FUNCTION_BLOCK "FB_DigitalOutputs"   // FB212, SCL
{ S7_Optimized_Access := 'TRUE' }
// stored: AutoNumber false, MemoryReserve 100, SetENOAutomatically false
   VAR
      sFreeQ0_0 : "FB_DigitalOutput";
      sOperatingCounter : "FB_DigitalOutput";
      sGeneralAirValve : "FB_DigitalOutput";
      sSmartLineDisable : "FB_DigitalOutput";
      sMachineLight : "FB_DigitalOutput";
      sMachineLightBack : "FB_DigitalOutput";
      sLightTowerOrange : "FB_DigitalOutput";
      sLightTowerRed : "FB_DigitalOutput";
      sLightTowerBlue : "FB_DigitalOutput";
      sLightTowerGreen : "FB_DigitalOutput";
      sLightTowerWhite : "FB_DigitalOutput";
      sBacklight : "FB_DigitalOutput";
      sFreeQ1_4 : "FB_DigitalOutput";
      sInfeedON : "FB_DigitalOutput";
      sAxisActivation : "FB_DigitalOutput";
      sBuzzerActivation : "FB_DigitalOutput";
      sElbaronPowerON : "FB_DigitalOutput";
      sObservationCameraLight : "FB_DigitalOutput";
      sLaserExternalDoorOpening : "FB_DigitalOutput";
      sCoolingStart : "FB_DigitalOutput";
      sX_AxisBrakeActivation : "FB_DigitalOutput";
      sY_AxisBrakeActivation : "FB_DigitalOutput";
      sAxisB_TeachInClampingPart : "FB_DigitalOutput";
      sEPO_UPS : "FB_DigitalOutput";
      sHeadLaserStart : "FB_DigitalOutput";
      sHeadLaserStop : "FB_DigitalOutput";
      sAxis2_PowerContactor : "FB_DigitalOutput";
      sGasAssistOn : "FB_DigitalOutput";
      sSmartLineReset : "FB_DigitalOutput";
      sXY_AxisPowerContactor : "FB_DigitalOutput";
      sLaserAirPressureProcess : "FB_DigitalOutput";
      sBus60V_PowerContactor : "FB_DigitalOutput";
      sFreeQ4_0 : "FB_DigitalOutput";
      sFreeQ4_1 : "FB_DigitalOutput";
      sFreeQ4_2 : "FB_DigitalOutput";
      sFreeQ4_3 : "FB_DigitalOutput";
      sLoadClampClosing : "FB_DigitalOutput";
      sLoadClampOpening : "FB_DigitalOutput";
      sUnloadClampClosing : "FB_DigitalOutput";
      sUnloadClampOpening : "FB_DigitalOutput";
      sClampingOpening : "FB_DigitalOutput";
      sClampingClosing : "FB_DigitalOutput";
      sB_AxisBrakeRelease : "FB_DigitalOutput";
      sSuction : "FB_DigitalOutput";
      sFreeQ5_4 : "FB_DigitalOutput";
      sFreeQ5_5 : "FB_DigitalOutput";
      sFreeQ5_6 : "FB_DigitalOutput";
      sFreeQ5_7 : "FB_DigitalOutput";
      sExternalGateClosing : "FB_DigitalOutput";
      sExternalGateOpening : "FB_DigitalOutput";
      sInternalGateClosing : "FB_DigitalOutput";
      sInternalGateOpening : "FB_DigitalOutput";
      sPowerMeterRetract : "FB_DigitalOutput";
      sPowerMeterAdvance : "FB_DigitalOutput";
      sBlowing : "FB_DigitalOutput";
      sFreeQ8_7 : "FB_DigitalOutput";
      sFreeQ9_0 : "FB_DigitalOutput";
      sFreeQ9_1 : "FB_DigitalOutput";
      sFreeQ9_2 : "FB_DigitalOutput";
      sFreeQ9_3 : "FB_DigitalOutput";
      sFreeQ9_4 : "FB_DigitalOutput";
      sFreeQ9_5 : "FB_DigitalOutput";
      sFreeQ9_6 : "FB_DigitalOutput";
      sFreeQ9_7 : "FB_DigitalOutput";
      sSonplasDiagDPCoupler { S7_SetPoint := 'True'} : "FB_DigitalOutput";
      sSonplasReady { S7_SetPoint := 'True'} : "FB_DigitalOutput";
      sSonplasNoEStop { S7_SetPoint := 'True'} : "FB_DigitalOutput";
      sSonplasDoorsClosed { S7_SetPoint := 'True'} : "FB_DigitalOutput";
      sSonplasRunError { S7_SetPoint := 'True'} : "FB_DigitalOutput";
      sSonplasFreeQ200_5 { S7_SetPoint := 'True'} : "FB_DigitalOutput";
      sSonplasFreeQ200_6 { S7_SetPoint := 'True'} : "FB_DigitalOutput";
      sSonplasFreeQ200_7 { S7_SetPoint := 'True'} : "FB_DigitalOutput";
      sSonplasFreeQ201_0 { S7_SetPoint := 'True'} : "FB_DigitalOutput";
      sSonplasFreeQ201_1 { S7_SetPoint := 'True'} : "FB_DigitalOutput";
      sSonplasFreeQ201_2 { S7_SetPoint := 'True'} : "FB_DigitalOutput";
      sSonplasFreeQ201_3 { S7_SetPoint := 'True'} : "FB_DigitalOutput";
      sSonplasFreeQ201_4 { S7_SetPoint := 'True'} : "FB_DigitalOutput";
      sSonplasFreeQ201_5 { S7_SetPoint := 'True'} : "FB_DigitalOutput";
      sSonplasFreeQ201_6 { S7_SetPoint := 'True'} : "FB_DigitalOutput";
      sSonplasFreeQ201_7 { S7_SetPoint := 'True'} : "FB_DigitalOutput";
      sSonplasShuttle1InPos { S7_SetPoint := 'True'} : "FB_DigitalOutput";
      sSonplasFreeQ202_1 { S7_SetPoint := 'True'} : "FB_DigitalOutput";
      sSonplasFreeQ202_2 { S7_SetPoint := 'True'} : "FB_DigitalOutput";
      sSonplasFreeQ202_3 { S7_SetPoint := 'True'} : "FB_DigitalOutput";
      sSonplasFreeQ202_4 { S7_SetPoint := 'True'} : "FB_DigitalOutput";
      sSonplasFreeQ202_5 { S7_SetPoint := 'True'} : "FB_DigitalOutput";
      sSonplasPart1OK { S7_SetPoint := 'True'} : "FB_DigitalOutput";
      sSonplasPart1NOK { S7_SetPoint := 'True'} : "FB_DigitalOutput";
      sSonplasShuttle2InPos { S7_SetPoint := 'True'} : "FB_DigitalOutput";
      sSonplasFreeQ203_1 { S7_SetPoint := 'True'} : "FB_DigitalOutput";
      sSonplasFreeQ203_2 { S7_SetPoint := 'True'} : "FB_DigitalOutput";
      sSonplasFreeQ203_3 { S7_SetPoint := 'True'} : "FB_DigitalOutput";
      sSonplasFreeQ203_4 { S7_SetPoint := 'True'} : "FB_DigitalOutput";
      sSonplasFreeQ203_5 { S7_SetPoint := 'True'} : "FB_DigitalOutput";
      sSonplasPart2OK { S7_SetPoint := 'True'} : "FB_DigitalOutput";
      sSonplasPart2NOK { S7_SetPoint := 'True'} : "FB_DigitalOutput";
      sSonplasResultAccepted { S7_SetPoint := 'True'} : "FB_DigitalOutput";
      sSonplasFreeQ244_1 { S7_SetPoint := 'True'} : "FB_DigitalOutput";
      sSonplasFreeQ244_2 { S7_SetPoint := 'True'} : "FB_DigitalOutput";
      sSonplasFreeQ244_3 { S7_SetPoint := 'True'} : "FB_DigitalOutput";
      sSonplasFreeQ244_4 { S7_SetPoint := 'True'} : "FB_DigitalOutput";
      sSonplasFreeQ244_5 { S7_SetPoint := 'True'} : "FB_DigitalOutput";
      sSonplasFreeQ244_6 { S7_SetPoint := 'True'} : "FB_DigitalOutput";
      sSonplasFreeQ244_7 { S7_SetPoint := 'True'} : "FB_DigitalOutput";
   END_VAR
BEGIN
   REGION Description head
       //==================================================================================
       // POSALUX Swiss SA / (C) Copyright 2025
       //----------------------------------------------------------------------------------
       // Title: Digital Ouputs mapping
       // Comment/Function: Digital Ouputs mapping
       // Author: Fabien WALDT
       // Engineering: TIA Portal v17
       //----------------------------------------------------------------------------------
       // Change log table:
       // Version  | Date     | Expert in charge | Changes applied
       //----------------------------------------------------------------------------------
       // 00.00.01 | 20250423 | WFA              | First released version
       //==================================================================================
   END_REGION


       // ET200SP Mapping
   REGION Q0.0 - Q1.7 : DQ 16x24VDC/0.5A ST Slot 5
       #sFreeQ0_0(oHWStatus => "DQ_FreeQ0_0");
       #sOperatingCounter(oHWStatus => "DQ_OperatingCounter");
       #sGeneralAirValve(oHWStatus => "DQ_GeneralAirValve");
       #sSmartLineDisable(oHWStatus => "DQ_SmartLineDisable");
       #sMachineLight(oHWStatus => "DQ_MachineLight");
       #sMachineLightBack(oHWStatus => "DQ_MachineLightBack");
       #sLightTowerOrange(oHWStatus => "DQ_LightTowerOrange");
       #sLightTowerRed(oHWStatus => "DQ_LightTowerRed");
       //
       #sLightTowerBlue(oHWStatus => "DQ_LightTowerBlue");
       #sLightTowerGreen(oHWStatus => "DQ_Light_owerGreen");
       #sLightTowerWhite(oHWStatus => "DQ_LightTowerWhite");
       #sBacklight(oHWStatus => "DQ_Backlight");
       #sFreeQ1_4(oHWStatus => "DQ_FreeQ1_4");
       #sInfeedON(oHWStatus => "DQ_InfeedON");
       #sAxisActivation(oHWStatus => "DQ_AxisActivation");
       #sBuzzerActivation(oHWStatus => "DQ_BuzzerActivation");
   END_REGION

   REGION Q2.0 - Q3.7 : DQ 16x24VDC/0.5A ST Slot 6
       #sElbaronPowerON(oHWStatus => "DQ_ElbaronPowerON");
       #sObservationCameraLight(oHWStatus => "DQ_ObservationCameraLight");
       #sLaserExternalDoorOpening(oHWStatus => "DQ_LaserExternalDoorOpening");
       #sCoolingStart(oHWStatus => "DQ_CoolingStart");
       #sX_AxisBrakeActivation(oHWStatus => "DQ_X_AxisBrakeActivation");
       #sY_AxisBrakeActivation(oHWStatus => "DQ_Y_AxisBrakeActivation");
       #sAxisB_TeachInClampingPart(oHWStatus => "DQ_AxisB_TeachInClampingPart");
       #sEPO_UPS(oHWStatus => "DQ_EPO_UPS");
       //
       #sHeadLaserStart(oHWStatus => "DQ_HeadLaserStart");
       #sHeadLaserStop(oHWStatus => "DQ_HeadLaserStop");
       #sAxis2_PowerContactor(oHWStatus => "DQ_Axis2_PowerContactor");
       #sGasAssistOn(oHWStatus => "DQ_GasAssistOn");
       #sSmartLineReset(oHWStatus => "DQ_SmartLineReset");
       #sXY_AxisPowerContactor(oHWStatus => "DQ_XY_AxisPowerContactor");
       #sLaserAirPressureProcess(oHWStatus => "DQ_LaserAirPressureProcess");
       #sBus60V_PowerContactor(oHWStatus => "DQ_Bus60V_PowerContactor");
   END_REGION

   REGION Q4.0 - Q5.7 : DQ 16x24VDC/0.5A ST Slot 7
       #sFreeQ4_0(oHWStatus => "DQ_FreeQ4_0");
       #sFreeQ4_1(oHWStatus => "DQ_FreeQ4_1");
       #sFreeQ4_2(oHWStatus => "DQ_FreeQ4_2");
       #sFreeQ4_3(oHWStatus => "DQ_FreeQ4_3");
       #sLoadClampClosing(oHWStatus => "DQ_LoadClampClosing");
       #sLoadClampOpening(oHWStatus => "DQ_LoadClampOpening");
       #sUnloadClampClosing(oHWStatus => "DQ_UnloadClampClosing");
       #sUnloadClampOpening(oHWStatus => "DQ_UnloadClampOpening");
       //
       #sClampingOpening(oHWStatus => "DQ_ClampingOpening");
       #sClampingClosing(oHWStatus => "DQ_ClampingClosing");
       #sB_AxisBrakeRelease(oHWStatus => "DQ_B_AxisBrakeRelease");
       #sSuction(oHWStatus => "DQ_Suction");
       #sFreeQ5_4(oHWStatus => "DQ_FreeQ5_4");
       #sFreeQ5_5(oHWStatus => "DQ_FreeQ5_5");
       #sFreeQ5_6(oHWStatus => "DQ_FreeQ5_6");
       #sFreeQ5_7(oHWStatus => "DQ_FreeQ5_7");
   END_REGION

   REGION Q8.0 - Q9.7 : DQ 16x24VDC/0.5A ST Slot 8
       #sExternalGateClosing(oHWStatus => "DQ_ExternalGateClosing");
       #sExternalGateOpening(oHWStatus => "DQ_ExternalGateOpening");
       #sInternalGateClosing(oHWStatus => "DQ_InternalGateClosing");
       #sInternalGateOpening(oHWStatus => "DQ_InternalGateOpening");
       #sPowerMeterRetract(oHWStatus => "DQ_PowerMeterRetract");
       #sPowerMeterAdvance(oHWStatus => "DQ_PowerMeterAdvance");
       #sBlowing(oHWStatus => "DQ_Blowing");
       #sFreeQ8_7(oHWStatus => "DQ_FreeQ8_7");
       //
       #sFreeQ9_0(oHWStatus => "DQ_FreeQ9_0");
       #sFreeQ9_1(oHWStatus => "DQ_FreeQ9_1");
       #sFreeQ9_2(oHWStatus => "DQ_FreeQ9_2");
       #sFreeQ9_3(oHWStatus => "DQ_FreeQ9_3");
       #sFreeQ9_4(oHWStatus => "DQ_FreeQ9_4");
       #sFreeQ9_5(oHWStatus => "DQ_FreeQ9_5");
       #sFreeQ9_6(oHWStatus => "DQ_FreeQ9_6");
       #sFreeQ9_7(oHWStatus => "DQ_FreeQ9_7");
   END_REGION
END_FUNCTION_BLOCK

FUNCTION_BLOCK "FB_DigitalOutput"   // FB32, SCL
{ S7_Optimized_Access := 'TRUE' }
// stored: AutoNumber false, MemoryReserve 100, SetENOAutomatically false
   VAR_OUTPUT
      oHWStatus : Bool;
   END_VAR
   VAR
      sSWStatus { ExternalAccessible := 'False'; ExternalVisible := 'False'; ExternalWritable := 'False'} : Bool;
      sHWStatus { ExternalAccessible := 'False'; ExternalVisible := 'False'; ExternalWritable := 'False'} : Bool;
   END_VAR
BEGIN
   REGION Description header 
       //==================================================================================
       // POSALUX Swiss SA / (C) Copyright 2024
       //----------------------------------------------------------------------------------
       // Title: Fonction Sortie Numérique
       // Comment/Function: This function handles the state of a PLC digital output.
       //                   It updates the hardware output state based on the software
       //                   state and assigns this state to the PLC's physical output.
       // Author: Gowsigan SRITHARAN
       // Engineering: TIA Portal v17
       //----------------------------------------------------------------------------------
       // Change log table:
       // Version  | Date     | Expert in charge | Changes applied
       // ---------|----------|------------------|------------------------------------
       // 00.00.01 | 20250106 | GSR              | First released version
       // ==================================================================================
   END_REGION

   REGION Hardware State Update
       #sHWStatus := #sSWStatus;
   END_REGION

   REGION Physical Output Assignment
       #oHWStatus := #sHWStatus;
   END_REGION
END_FUNCTION_BLOCK

FUNCTION_BLOCK "FB_DigitalOutputsSonplas"   // FB213, SCL
{ S7_Optimized_Access := 'TRUE' }
// stored: AutoNumber false, MemoryReserve 100, SetENOAutomatically false
   VAR
      Free_Q0_0 : "FB_DigitalOutput";
      Operating_Counter : "FB_DigitalOutput";
      General_Air_Valve : "FB_DigitalOutput";
      Smart_Line_Disable : "FB_DigitalOutput";
      Machine_Light : "FB_DigitalOutput";
      Machine_Light_Back : "FB_DigitalOutput";
      Light_Tower_Orange : "FB_DigitalOutput";
      Light_Tower_Red : "FB_DigitalOutput";
      Light_Tower_Blue : "FB_DigitalOutput";
      Light_Tower_Green : "FB_DigitalOutput";
      Light_Tower_White : "FB_DigitalOutput";
      Backlight : "FB_DigitalOutput";
      Free_Q1_4 : "FB_DigitalOutput";
      Infeed_ON : "FB_DigitalOutput";
      Axis_Activation : "FB_DigitalOutput";
      Buzzer_Activation : "FB_DigitalOutput";
      Elbaron_Power_ON : "FB_DigitalOutput";
      Observation_Camera_Light : "FB_DigitalOutput";
      Laser_External_Door_Opening : "FB_DigitalOutput";
      Cooling_Start : "FB_DigitalOutput";
      X_Axis_Brake_Activation : "FB_DigitalOutput";
      Y_Axis_Brake_Activation : "FB_DigitalOutput";
      Axis_B_TeachIn_Clamping_Part : "FB_DigitalOutput";
      EPO_UPS : "FB_DigitalOutput";
      Head_Laser_Start : "FB_DigitalOutput";
      Head_Laser_Stop : "FB_DigitalOutput";
      Axis_2_Power_Contactor : "FB_DigitalOutput";
      GasAssistOn : "FB_DigitalOutput";
      Smart_Line_Reset : "FB_DigitalOutput";
      XY_Axis_Power_Contactor : "FB_DigitalOutput";
      Laser_Air_Pressure_Process : "FB_DigitalOutput";
      Bus60V_Power_Contactor : "FB_DigitalOutput";
      Free_Q4_0 : "FB_DigitalOutput";
      Free_Q4_1 : "FB_DigitalOutput";
      Free_Q4_2 : "FB_DigitalOutput";
      Free_Q4_3 : "FB_DigitalOutput";
      Load_Clamp_Closing : "FB_DigitalOutput";
      Load_Clamp_Opening : "FB_DigitalOutput";
      Unload_Clamp_Closing : "FB_DigitalOutput";
      Unload_Clamp_Opening : "FB_DigitalOutput";
      Clamping_Opening : "FB_DigitalOutput";
      Clamping_Closing : "FB_DigitalOutput";
      B_Axis_Brake_Release : "FB_DigitalOutput";
      Suction : "FB_DigitalOutput";
      Free_Q5_4 : "FB_DigitalOutput";
      Free_Q5_5 : "FB_DigitalOutput";
      Free_Q5_6 : "FB_DigitalOutput";
      Free_Q5_7 : "FB_DigitalOutput";
      External_Gate_Closing : "FB_DigitalOutput";
      External_Gate_Opening : "FB_DigitalOutput";
      Internal_Gate_Closing : "FB_DigitalOutput";
      Internal_Gate_Opening : "FB_DigitalOutput";
      PowerMeter_Retract : "FB_DigitalOutput";
      PowerMeter_Advance : "FB_DigitalOutput";
      Blowing : "FB_DigitalOutput";
      Free_Q8_7 : "FB_DigitalOutput";
      Free_Q9_0 : "FB_DigitalOutput";
      Free_Q9_1 : "FB_DigitalOutput";
      Free_Q9_2 : "FB_DigitalOutput";
      Free_Q9_3 : "FB_DigitalOutput";
      Free_Q9_4 : "FB_DigitalOutput";
      Free_Q9_5 : "FB_DigitalOutput";
      Free_Q9_6 : "FB_DigitalOutput";
      Free_Q9_7 : "FB_DigitalOutput";
      Sonplas_DiagDPCoupler { S7_SetPoint := 'True'} : "FB_DigitalOutput";
      Sonplas_Ready { S7_SetPoint := 'True'} : "FB_DigitalOutput";
      Sonplas_NoEStop { S7_SetPoint := 'True'} : "FB_DigitalOutput";
      Sonplas_DoorsClosed { S7_SetPoint := 'True'} : "FB_DigitalOutput";
      Sonplas_RunError { S7_SetPoint := 'True'} : "FB_DigitalOutput";
      Sonplas_Free_Q200_5 { S7_SetPoint := 'True'} : "FB_DigitalOutput";
      Sonplas_Free_Q200_6 { S7_SetPoint := 'True'} : "FB_DigitalOutput";
      Sonplas_Free_Q200_7 { S7_SetPoint := 'True'} : "FB_DigitalOutput";
      Sonplas_Free_Q201_0 { S7_SetPoint := 'True'} : "FB_DigitalOutput";
      Sonplas_Free_Q201_1 { S7_SetPoint := 'True'} : "FB_DigitalOutput";
      Sonplas_Free_Q201_2 { S7_SetPoint := 'True'} : "FB_DigitalOutput";
      Sonplas_Free_Q201_3 { S7_SetPoint := 'True'} : "FB_DigitalOutput";
      Sonplas_Free_Q201_4 { S7_SetPoint := 'True'} : "FB_DigitalOutput";
      Sonplas_Free_Q201_5 { S7_SetPoint := 'True'} : "FB_DigitalOutput";
      Sonplas_Free_Q201_6 { S7_SetPoint := 'True'} : "FB_DigitalOutput";
      Sonplas_Free_Q201_7 { S7_SetPoint := 'True'} : "FB_DigitalOutput";
      Sonplas_Shuttle1InPos { S7_SetPoint := 'True'} : "FB_DigitalOutput";
      Sonplas_Free_Q202_1 { S7_SetPoint := 'True'} : "FB_DigitalOutput";
      Sonplas_Free_Q202_2 { S7_SetPoint := 'True'} : "FB_DigitalOutput";
      Sonplas_Free_Q202_3 { S7_SetPoint := 'True'} : "FB_DigitalOutput";
      Sonplas_Free_Q202_4 { S7_SetPoint := 'True'} : "FB_DigitalOutput";
      Sonplas_Free_Q202_5 { S7_SetPoint := 'True'} : "FB_DigitalOutput";
      Sonplas_Part1OK { S7_SetPoint := 'True'} : "FB_DigitalOutput";
      Sonplas_Part1NOK { S7_SetPoint := 'True'} : "FB_DigitalOutput";
      Sonplas_Shuttle2InPos { S7_SetPoint := 'True'} : "FB_DigitalOutput";
      Sonplas_Free_Q203_1 { S7_SetPoint := 'True'} : "FB_DigitalOutput";
      Sonplas_Free_Q203_2 { S7_SetPoint := 'True'} : "FB_DigitalOutput";
      Sonplas_Free_Q203_3 { S7_SetPoint := 'True'} : "FB_DigitalOutput";
      Sonplas_Free_Q203_4 { S7_SetPoint := 'True'} : "FB_DigitalOutput";
      Sonplas_Free_Q203_5 { S7_SetPoint := 'True'} : "FB_DigitalOutput";
      Sonplas_Part2OK { S7_SetPoint := 'True'} : "FB_DigitalOutput";
      Sonplas_Part2NOK { S7_SetPoint := 'True'} : "FB_DigitalOutput";
      Sonplas_ResultAccepted { S7_SetPoint := 'True'} : "FB_DigitalOutput";
      Sonplas_Free_Q244_1 { S7_SetPoint := 'True'} : "FB_DigitalOutput";
      Sonplas_Free_Q244_2 { S7_SetPoint := 'True'} : "FB_DigitalOutput";
      Sonplas_Free_Q244_3 { S7_SetPoint := 'True'} : "FB_DigitalOutput";
      Sonplas_Free_Q244_4 { S7_SetPoint := 'True'} : "FB_DigitalOutput";
      Sonplas_Free_Q244_5 { S7_SetPoint := 'True'} : "FB_DigitalOutput";
      Sonplas_Free_Q244_6 { S7_SetPoint := 'True'} : "FB_DigitalOutput";
      Sonplas_Free_Q244_7 { S7_SetPoint := 'True'} : "FB_DigitalOutput";
   END_VAR
BEGIN
   REGION Description head
       //==================================================================================
       // POSALUX Swiss SA / (C) Copyright 2025
       //----------------------------------------------------------------------------------
       // Title: Digital Ouputs mapping
       // Comment/Function: Sonplas Digital Ouputs mapping
       // Author: Fabien WALDT
       // Engineering: TIA Portal v17
       //----------------------------------------------------------------------------------
       // Change log table:
       // Version  | Date     | Expert in charge | Changes applied
       //----------------------------------------------------------------------------------
       // 00.00.01 | 20250423 | WFA              | First released version
       //==================================================================================
   END_REGION

   REGION Operating modes AND parts exchange
       #Sonplas_DiagDPCoupler(oHWStatus => "DQ_SonplasDiagDPCoupler");
       #Sonplas_Ready(oHWStatus => "DQ_SonplasReady");
       #Sonplas_NoEStop(oHWStatus => "DQ_SonplasNoEStop");
       #Sonplas_DoorsClosed(oHWStatus => "DQ_SonplasDoorsClosed");
       #Sonplas_RunError(oHWStatus => "DQ_SonplasRunError");
       #Sonplas_Free_Q200_5(oHWStatus => "DQ_SonplasFreeQ200_5");
       #Sonplas_Free_Q200_6(oHWStatus => "DQ_SonplasFreeQ200_6");
       #Sonplas_Free_Q200_7(oHWStatus => "DQ_SonplasFreeQ200_7");
       // 
       #Sonplas_Free_Q201_0(oHWStatus => "DQ_SonplasFreeQ201_0");
       #Sonplas_Free_Q201_1(oHWStatus => "DQ_SonplasFreeQ201_1");
       #Sonplas_Free_Q201_2(oHWStatus => "DQ_SonplasFreeQ201_2");
       #Sonplas_Free_Q201_3(oHWStatus => "DQ_SonplasFreeQ201_3");
       #Sonplas_Free_Q201_4(oHWStatus => "DQ_SonplasFreeQ201_4");
       #Sonplas_Free_Q201_5(oHWStatus => "DQ_SonplasFreeQ201_5");
       #Sonplas_Free_Q201_6(oHWStatus => "DQ_SonplasFreeQ201_6");
       #Sonplas_Free_Q201_7(oHWStatus => "DQ_SonplasFreeQ201_7");
   END_REGION

   REGION Part exchange
       #Sonplas_Shuttle1InPos(oHWStatus => "DQ_SonplasShuttle1InPos");
       #Sonplas_Free_Q202_1(oHWStatus => "DQ_SonplasFreeQ202_1");
       #Sonplas_Free_Q202_2(oHWStatus => "DQ_SonplasFreeQ202_2");
       #Sonplas_Free_Q202_3(oHWStatus => "DQ_SonplasFreeQ202_3");
       #Sonplas_Free_Q202_4(oHWStatus => "DQ_SonplasFreeQ202_4");
       #Sonplas_Free_Q202_5(oHWStatus => "DQ_SonplasFreeQ202_5");
       #Sonplas_Part1OK(oHWStatus => "DQ_SonplasPart1OK");
       #Sonplas_Part1NOK(oHWStatus => "DQ_SonplasPart1NOK");
       // 
       #Sonplas_Shuttle2InPos(oHWStatus => "DQ_SonplasShuttle2InPos");
       #Sonplas_Free_Q203_1(oHWStatus => "DQ_SonplasFreeQ203_1");
       #Sonplas_Free_Q203_2(oHWStatus => "DQ_SonplasFreeQ203_2");
       #Sonplas_Free_Q203_3(oHWStatus => "DQ_SonplasFreeQ203_3");
       #Sonplas_Free_Q203_4(oHWStatus => "DQ_SonplasFreeQ203_4");
       #Sonplas_Free_Q203_5(oHWStatus => "DQ_SonplasFreeQ203_5");
       #Sonplas_Part2OK(oHWStatus => "DQ_SonplasPart2OK");
       #Sonplas_Part2NOK(oHWStatus => "DQ_SonplasPart2NOK");
   END_REGION

   REGION Measure
       #Sonplas_ResultAccepted(oHWStatus => "DQ_SonplasResultAccepted");
       #Sonplas_Free_Q244_1(oHWStatus => "DQ_SonplasFreeQ244_1");
       #Sonplas_Free_Q244_2(oHWStatus => "DQ_SonplasFreeQ244_2");
       #Sonplas_Free_Q244_3(oHWStatus => "DQ_SonplasFreeQ244_3");
       #Sonplas_Free_Q244_4(oHWStatus => "DQ_SonplasFreeQ244_4");
       #Sonplas_Free_Q244_5(oHWStatus => "DQ_SonplasFreeQ244_5");
       #Sonplas_Free_Q244_6(oHWStatus => "DQ_SonplasFreeQ244_6");
       #Sonplas_Free_Q244_7(oHWStatus => "DQ_SonplasFreeQ244_7");
   END_REGION
END_FUNCTION_BLOCK

FUNCTION_BLOCK "FB_Impulsion"   // FB52, SCL
{ S7_Optimized_Access := 'TRUE' }
// stored: MemoryReserve 100, SetENOAutomatically false
   VAR RETAIN
      sCountSecPulseMinute : DInt;
      sCountSecPulseHour : DInt;
      sCountSecPulseDay : DInt;
   END_VAR
   VAR
      sPulseMinute : Bool;   // Impulsion every minute
      sPulseHour : Bool;   // Impulsion every hour
      sPulseDay : Bool;   // Impulsion every day
      sRT_Clock_1Hz { S7_SetPoint := 'True'} : R_TRIG;
   END_VAR
   VAR CONSTANT
      MAX_COUNT_MINUTE : DInt := 60;
      MAX_COUNT_HOUR : DInt := 3600;
      MAX_COUNT_DAY : DInt := 86400;
   END_VAR
BEGIN
   REGION Description header 
       //==================================================================================
       // POSALUX Swiss SA / (C) Copyright 2024
       //----------------------------------------------------------------------------------
       // Title: Time counter
       // Comment/Function: Generates periodic pulses using 1Hz clock base
       //                      - Minute interval pulses (60s cycle)
       //                      - Hour interval pulses (3600s cycle)
       //                      - Day interval pulses (86400s cycle)
       //                   Implementation: Uses cascaded counters with 1Hz clock input
       // Author: Gowsigan SRITHARAN
       // Engineering: TIA Portal v17
       //----------------------------------------------------------------------------------
       // Change log table:
       // Version  | Date     | Expert in charge | Changes applied
       // ---------|----------|------------------|------------------------------------
       // 00.00.01 | 20241206 | GSR              | First released version
       // ---------|----------|------------------|------------------------------------
       // 01.01.01 | 20241219 | FMI              | Utilisation d'un flanc montant du clock1Hz pour compter en secondes
       // ==================================================================================
   END_REGION

   REGION Rising edge detection and counter incrementation
       #sRT_Clock_1Hz.CLK:="Clock_1Hz";
       #sRT_Clock_1Hz();
     IF  #sRT_Clock_1Hz.Q THEN
       #sCountSecPulseMinute := #sCountSecPulseMinute + 1;
       #sCountSecPulseHour := #sCountSecPulseHour + 1;
       #sCountSecPulseDay := #sCountSecPulseDay + 1;
   END_IF;
   END_REGION

   REGION Pulse generation and counter reset
       // Impulsion minute
       IF #sCountSecPulseMinute >= #MAX_COUNT_MINUTE THEN
           #sPulseMinute := TRUE;
           #sCountSecPulseMinute := 0;
       ELSE
           #sPulseMinute := FALSE;
       END_IF;

       // Impulsion hour
       IF #sCountSecPulseHour >= #MAX_COUNT_HOUR THEN
           #sPulseHour := TRUE;
           #sCountSecPulseHour := 0;
       ELSE
           #sPulseHour := FALSE;
       END_IF;

       // Impulsion day
       IF #sCountSecPulseDay >= #MAX_COUNT_DAY THEN
           #sPulseDay := TRUE;
           #sCountSecPulseDay := 0;
       ELSE
           #sPulseDay := FALSE;
       END_IF;
   END_REGION
END_FUNCTION_BLOCK

FUNCTION_BLOCK "FB_ReadDateAndTime"   // FB46, SCL
{ S7_Optimized_Access := 'TRUE' }
// stored: MemoryReserve 100, SetENOAutomatically false
   VAR
      sDateAndTime : DTL;
      sCurrentDT : Struct
         sYear : UInt;
         sMonth : USInt;
         sDay : USInt;
         sHour : USInt;
         sMinute : USInt;
         sSecond : USInt;
         sNanoSecond : UDInt;
      END_STRUCT;
   END_VAR
   VAR_TEMP
      tRetVal : Int;
   END_VAR
BEGIN
   REGION Description header 
       //==================================================================================
       // POSALUX Swiss SA / (C) Copyright 2025
       //----------------------------------------------------------------------------------
       // Title: FB_ReadDateAndTime
       // Comment/Function: Reading the date and time of the PLC
       // Author: Fabien WALDT
       // Engineering: TIA Portal v20
       //----------------------------------------------------------------------------------
       // Change log table:
       // Version  | Date     | Expert in charge | Changes applied
       // ---------|----------|------------------|-----------------------------------------
       // 00.00.01 | 20251017 | WFA              | First released version
       // =================================================================================
   END_REGION

   REGION Lecture Date et Heure
       #tRetVal :=RD_SYS_T(OUT => #sDateAndTime);
       #sCurrentDT.sYear       := #sDateAndTime.YEAR;
       #sCurrentDT.sMonth      := #sDateAndTime.MONTH;
       #sCurrentDT.sHour      := #sDateAndTime.HOUR;
       #sCurrentDT.sMinute     := #sDateAndTime.MINUTE;
       #sCurrentDT.sSecond     := #sDateAndTime.SECOND;
       #sCurrentDT.sNanoSecond := #sDateAndTime.NANOSECOND;
   END_REGION
END_FUNCTION_BLOCK

FUNCTION_BLOCK "FB_CommPLC_ISO"   // FB1100, SCL
{ S7_Optimized_Access := 'TRUE' }
// stored: AutoNumber false, MemoryReserve 100, SetENOAutomatically false
   VAR DB_SPECIFIC
      sSynchro_ULx { ExternalVisible := 'False'; ExternalWritable := 'False'} : Byte;   // Image of A_DBB[1000]
   END_VAR
   VAR
      sSynchro_ULx_WriteON { ExternalAccessible := 'False'; ExternalVisible := 'False'; ExternalWritable := 'False'} : Bool;
      sRT_FixtureVW_Rel : R_TRIG;
      sRT_FixtureVW_Req { S7_SetPoint := 'True'} : R_TRIG;
      sRT_GripperAvail { S7_SetPoint := 'True'} : R_TRIG;
      sAxisManagedByNC { S7_SetPoint := 'True'} : Bool;
      sAxisReservedbyNC : Bool;
   END_VAR
   VAR_TEMP
      tSynchro_ULx_ReadON : Bool;
      tReadError : Bool;
      tWriteError : Bool;
      tReadErrCode : Int;
      tWriteErrCode : Int;
   END_VAR
BEGIN

   REGION Read/Write Byte Cmd : $A_DBB[1000]
       // SYNCHRO_UL1
       // SYNCHRO_UL1 = 1 : Demande axes par NC (Mise à 1 par NC)
       // SYNCHRO_UL1 = 0 : Liberation axes par PLC (Mise à 0 par PLC)

       #sRT_GripperAvail(CLK := "DB_GestionGripper".sGripperStatus.Available);


       #sRT_FixtureVW_Req(CLK := (("DB_LoaderFixture".sFixtureMain.iGripperReadyForUnloading AND NOT "DB_WorkingModes".sFilling) // Gripper ready for Unloading
                          OR ("DB_LoaderFixture".sFixtureMain.iGripperReadyForLoading AND "DB_WorkingModes".sFilling)            // Gripper ready for Loading
                          OR #sRT_GripperAvail.Q                                                                                 // Gripper Available  
                          OR "DB_WorkingModes".sManu) AND #sSynchro_ULx.%X0);                                                    // Mode Manu
       IF #sRT_FixtureVW_Req.Q THEN
           #sSynchro_ULx.%X0 := FALSE;
           #sSynchro_ULx_WriteON := TRUE;
       END_IF;

       // SYNCHRO_UL2
       // SYNCHRO_UL2 = 1 : Liberation axes par NC (Mise à 1 par NC)
       // SYNCHRO_UL2 = 0 : Demande axes par PLC (Mise à 0 par PLC)   
       #sRT_FixtureVW_Rel(CLK := "DB_GestionGripper".sGripperStatus.Available AND #sSynchro_ULx.%X1); // Acquittement Liberation dès que Gripper Available
       IF #sRT_FixtureVW_Rel.Q THEN
           #sSynchro_ULx.%X1 := FALSE;
           #sSynchro_ULx_WriteON := TRUE;
       END_IF;

       // Axis reserved by NC
       IF #sRT_FixtureVW_Req.Q THEN
           #sAxisReservedbyNC := TRUE;
       ELSIF  #sRT_FixtureVW_Rel.Q OR "LBP_Chan1".A_Reset THEN
           #sAxisReservedbyNC := FALSE;
       END_IF;

       // Datas FOR Communication PLC <--> ISO
           // DEFINE xREAD_SYNCHRO_UL1         AS (($A_DBB[1000] B_AND 1)==1)
           // DEFINE xWRITE_ON_SYNCHRO_UL1     AS $A_DBB[1000]=$A_DBB[1000] B_OR 1
           // DEFINE xWRITE_OFF_SYNCHRO_UL1    AS $A_DBB[1000]=$A_DBB[1000] B_AND (255-1)

           // DEFINE xREAD_SYNCHRO_UL2         AS (($A_DBB[1000] B_AND 2)==2)
           // DEFINE xWRITE_ON_SYNCHRO_UL2     AS $A_DBB[1000]=$A_DBB[1000] B_OR 2
           // DEFINE xWRITE_OFF_SYNCHRO_UL2    AS $A_DBB[1000]=$A_DBB[1000] B_AND (255-2)
           // 


       // SYNCHRO_UL2 = 1 : Liberation axes par NC (Mise à 1 par NC)
       // SYNCHRO_UL2 = 0 : Demande axes par PLC (Mise à 0 par PLC)
       "LBP_TransferSelData"(Enable := #sSynchro_ULx_WriteON,
                             Funct := 4,
                             S7Var := #sSynchro_ULx,
                             IVAR1 := 1000,
                             IVAR2 := -1,
                             Error => #tWriteError,
                             ErrCode => #tWriteErrCode);

       IF NOT #sSynchro_ULx_WriteON THEN
           #tSynchro_ULx_ReadON := True;
       ELSE
           #tSynchro_ULx_ReadON := False;
       END_IF;
       IF (#sSynchro_ULx_WriteON AND NOT #tWriteError) THEN
           #sSynchro_ULx_WriteON := False;
       END_IF;

       "LBP_TransferSelData"(Enable := #tSynchro_ULx_ReadON,
                             Funct := 3,
                             S7Var := #sSynchro_ULx,
                             IVAR1 := 1000,
                             IVAR2 := -1,
                             Error => #tReadError,
                             ErrCode => #tReadErrCode);
   END_REGION
END_FUNCTION_BLOCK

FUNCTION_BLOCK "FB_MiscPLC_IHM_ISO"   // FB50, SCL
{ S7_Optimized_Access := 'TRUE' }
// stored: MemoryReserve 100, SetENOAutomatically false
   VAR
      sTransferSelData { S7_SetPoint := 'True'} : Array[0..11] of Byte;
      sTransferActData : Array[0..11] of Byte;
      sUpdate_PLC_ISO_Values : Bool;
      sRT_bStopAfterEmptying : R_TRIG;
      sRT_CNCModeReq { S7_SetPoint := 'True'} : R_TRIG;
   END_VAR
   VAR_TEMP
      tLoop : Int;
      tTransferSelDataError : Int;
      tTransferSelDataErrCode : Array[0..11] of Int;
   END_VAR
BEGIN
   REGION Description header 
       //==================================================================================
       // POSALUX Swiss SA / (C) Copyright 2025
       //----------------------------------------------------------------------------------
       // Title: 
       // Comment/Function: 
       // Author: Fabien WALDT
       // Engineering: TIA Portal v17
       //----------------------------------------------------------------------------------
       // Change log table:
       // Version  | Date     | Expert in charge | Changes applied
       // ---------|----------|------------------|-----------------------------------------
       // 00.00.01 | 20250423 | WFA              | First released version
       // =================================================================================
   END_REGION

   REGION Byte 960
       // Bit 0
       "DB_PLC_ISO_IHM".WarmUpOn := "LBP_AlarmMsgs".UserA[0].A70UUxx[35];

       // Bit 1
       "DB_PLC_ISO_IHM".KeyLaserOn := "DB_DataFromSafety".iKeyLaserOn;

       // Bit 2
       "DB_PLC_ISO_IHM".KeySaveParameters := "DB_McpKeyboardSignals".sK3_KeySaveParam.sKeySWToggleStatus;
       "DB_McpKeyboardSignals".sK3_KeySaveParam.sLedSWStatus := "DB_McpKeyboardSignals".sK3_KeySaveParam.sKeySWToggleStatus;

       // Bit 3
       // STOP_PROG_RUN est nommé bStopAfterEmptying dans PLC
       #sRT_bStopAfterEmptying(CLK := "DB_WorkingModes".sEmptying AND "DB_PartManagement".sPosition.sMachineEmpty);
       IF #sRT_bStopAfterEmptying.Q THEN
           "DB_PLC_ISO_IHM".bStopAfterEmptying := TRUE;
           "LBP_AlarmMsgs".UserA[0].A70UUxx[59] := TRUE;
           "DB_WorkingModes".sEmptying := FALSE;
           "DB_LoaderShuttle1".sMain.iJobReq := FALSE;
           "DB_LoaderShuttle2".sMain.iJobReq := FALSE;
       ELSIF "LBP_Chan1".E_ChanReset THEN
           "DB_PLC_ISO_IHM".bStopAfterEmptying := FALSE;
       END_IF;

       // Bit 4
       "DB_PLC_ISO_IHM".Chan1_running := "DB_CycleStartStop".sChan1Start;

       // Bit 5
       "DB_PLC_ISO_IHM".Chan2_running := FALSE;

       // Bit 6
       "DB_PLC_ISO_IHM".Chan3_running := FALSE;

       // Bit 7
       "DB_PLC_ISO_IHM".Chan4_running := FALSE;
   END_REGION

   REGION Byte 961
       // Bit 0
       "DB_PLC_ISO_IHM".StopAtNextReq := "DB_CycleStartStop".sResquestStopNextCycle;

       // Bit 1
       "DB_PLC_ISO_IHM".AllChanStop := NOT "DB_CycleStartStop".sChan1Start;

       // Bit 2
       "DB_PLC_ISO_IHM".LoaderAutomaticMode := "DB_WorkingModes".sAuto;

       // Bit 3
       "DB_PLC_ISO_IHM".LoaderManualMode := "DB_WorkingModes".sSemiAuto;

       // Bit 4 (NOT USED ON FL0125)
       "DB_PLC_ISO_IHM".NoCameraPresent := "DB_PLC_ISO_IHM".NoCameraPresent;

       // Bit 5 (NOT USED ON FL0125)
       "DB_PLC_ISO_IHM".PremeasureZexists := "DB_PLC_ISO_IHM".PremeasureZexists;

       // Bit 6 (NOT USED ON FL0125)
       "DB_PLC_ISO_IHM".PremeasureCexists := "DB_PLC_ISO_IHM".PremeasureCexists;

       // Bit 7
       "DB_PLC_ISO_IHM".PLCFunctNotFinished :=
       "DB_LoaderFixtureMain".sBlowingNotFinished
       OR "DB_LoaderFixtureMain".sLoadingNotFinished
       OR "DB_LoaderFixtureMain".sUnloadingNotFinished
       OR "DB_LoaderFixtureMain".sReleaseNotFinished
       OR "DB_LoaderFixtureMain".sV_InitNotFinished
       OR "DB_LoaderFixtureMain".sW_InitNotFinished;
   END_REGION

   REGION Byte 962
       // Bit 0
       // CAN_CHANGE_PART_LOADER_1 est nommé StartChangePart_station1 dans PLC
       #sRT_CNCModeReq(CLK := "DB_LoaderAxis".iCNCModeReq);

       IF #sRT_CNCModeReq.Q AND NOT "DB_PartManagement".sPosition.sMachineEmpty THEN
           "DB_PLC_ISO_IHM".StartChangePart_station1 := TRUE;
       ELSIF "LBP_Chan1".MDyn[76] THEN
           "DB_PLC_ISO_IHM".StartChangePart_station1 := FALSE;
       END_IF;

       // Bit 1
       "DB_PLC_ISO_IHM".StartCheckPart_fixture1 := "DB_PLC_ISO_IHM".StartCheckPart_fixture1;

       // Bit 2
       "DB_PLC_ISO_IHM".Loader1PartLoad := "DB_PartManagement".sPosition.sGripper.Undrilled.Presence.Part AND "DB_PartManagement".sPosition.sGripper.Undrilled.Presence.BW;

       // Bit 3
       "DB_PLC_ISO_IHM".Loader1PartUnload := "DB_PartManagement".sPosition.sGripper.Drilled.Presence.Part;

       // Bit 4
       "DB_PLC_ISO_IHM".Loader1ShiftLoad := "DB_PLC_ISO_IHM".Loader1ShiftLoad;

       // Bit 5
       "DB_PLC_ISO_IHM".Loader1ShiftUnload := "DB_PLC_ISO_IHM".Loader1ShiftUnload;

       // Bit 6
       "DB_PLC_ISO_IHM".Loader1LoadOpened := "DB_PLC_ISO_IHM".Loader1LoadOpened;

       // Bit 7
       "DB_PLC_ISO_IHM".Loader1UnloadOpened := "DB_PLC_ISO_IHM".Loader1UnloadOpened;
   END_REGION

   REGION Byte 963
       // Bit 0
       "DB_PLC_ISO_IHM".PartOnFixture1 := "DB_GestionFixture".sFixturePartControl.oGoodPart
               OR "DB_PartManagement".sPosition.sFixture.Undrilled.Presence.Part
               OR "DB_PartManagement".sPosition.sFixture.Drilled.Presence.Part;

       // Bit 1
       "DB_PLC_ISO_IHM".MasterOnFixture1 := "DB_PLC_ISO_IHM".MasterOnFixture1;

       // Bit 2
       "DB_PLC_ISO_IHM".StartChangePart_station2 := "DB_PLC_ISO_IHM".StartChangePart_station2;

       // Bit 3
       "DB_PLC_ISO_IHM".StartCheckPart_fixture2 := "DB_PLC_ISO_IHM".StartCheckPart_fixture2;

       // Bit 4
       "DB_PLC_ISO_IHM".Loader2PartLoad := "DB_PLC_ISO_IHM".Loader2PartLoad;

       // Bit 5
       "DB_PLC_ISO_IHM".Loader2PartUnload := "DB_PLC_ISO_IHM".Loader2PartUnload;

       // Bit 6
       "DB_PLC_ISO_IHM".Loader2ShiftLoad := "DB_PLC_ISO_IHM".Loader2ShiftLoad;

       // Bit 7
       "DB_PLC_ISO_IHM".Loader2ShiftUnload := "DB_PLC_ISO_IHM".Loader2ShiftUnload;
   END_REGION

   REGION Byte 964
       // Bit 0
       "DB_PLC_ISO_IHM".Loader2LoadOpened := "DB_PLC_ISO_IHM".Loader2LoadOpened;

       // Bit 1
       "DB_PLC_ISO_IHM".Loader2UnloadOpened := "DB_PLC_ISO_IHM".Loader2UnloadOpened;

       // Bit 2 
       "DB_PLC_ISO_IHM".PartOnFixture2 := "DB_PLC_ISO_IHM".PartOnFixture2;

       // Bit 3 (NOT USED ON FL0125)
       "DB_PLC_ISO_IHM".MasterOnFixture2 := "DB_PLC_ISO_IHM".MasterOnFixture2;

       // Bit 4 (NOT USED ON FL0125)
       "DB_PLC_ISO_IHM".StartChangePart_station3 := "DB_PLC_ISO_IHM".StartChangePart_station3;

       // Bit 5 (NOT USED ON FL0125)
       "DB_PLC_ISO_IHM".StartCheckPart_fixture3 := "DB_PLC_ISO_IHM".StartCheckPart_fixture3;

       // Bit 6 (NOT USED ON FL0125)
       "DB_PLC_ISO_IHM".Loader3PartLoad := "DB_PLC_ISO_IHM".Loader3PartLoad;

       // Bit 7 (NOT USED ON FL0125)
       "DB_PLC_ISO_IHM".Loader3PartUnload := "DB_PLC_ISO_IHM".Loader3PartUnload;
   END_REGION

   REGION Byte 965
       // Bit 0 (NOT USED ON FL0125)
       "DB_PLC_ISO_IHM".Loader3ShiftLoad := "DB_PLC_ISO_IHM".Loader3ShiftLoad;

       // Bit 1 (NOT USED ON FL0125)
       "DB_PLC_ISO_IHM".Loader3ShiftUnload := "DB_PLC_ISO_IHM".Loader3ShiftUnload;

       // Bit 2 (NOT USED ON FL0125)
       "DB_PLC_ISO_IHM".Loader3LoadOpened := "DB_PLC_ISO_IHM".Loader3LoadOpened;

       // Bit 3
       "DB_PLC_ISO_IHM".Loader3UnloadOpened := "DB_PLC_ISO_IHM".Loader3UnloadOpened;

       // Bit 4
       "DB_PLC_ISO_IHM".PartOnFixture3 := "DB_PLC_ISO_IHM".PartOnFixture3;

       // Bit 5 (NOT USED ON FL0125)
       "DB_PLC_ISO_IHM".MasterOnFixture3 := "DB_PLC_ISO_IHM".MasterOnFixture3;

       // Bit 6 (NOT USED ON FL0125)
       "DB_PLC_ISO_IHM".Part_KO_go_outside_mach := "DB_PLC_ISO_IHM".Part_KO_go_outside_mach;

       // Bit 7 (NOT USED ON FL0125)
       "DB_PLC_ISO_IHM".MasterOnMachine := "DB_PLC_ISO_IHM".MasterOnMachine;
   END_REGION

   REGION Word 968
       "DB_PLC_ISO_IHM".WarmUpTime := "DB_PLC_ISO_IHM".WarmUpTime;
   END_REGION

   REGION Byte 970
       // Bit 0
       "DB_PLC_ISO_IHM".Stop_For_BackWall_Wear_1 := "DB_PLC_ISO_IHM".Stop_For_BackWall_Wear_1;

       // Bit 1
       "DB_PLC_ISO_IHM".Stop_For_BackWall_Wear_2 := "DB_PLC_ISO_IHM".Stop_For_BackWall_Wear_2;

       // Bit 2
       "DB_PLC_ISO_IHM".Cleaning_Station_1 := "DB_PLC_ISO_IHM".Cleaning_Station_1;

       // Bit 3
       "DB_PLC_ISO_IHM".Cleaning_Station_2 := "DB_PLC_ISO_IHM".Cleaning_Station_2;

       // Bit 4
       "DB_PLC_ISO_IHM".Cleaning_Backwall_1 := "DB_PLC_ISO_IHM".Cleaning_Backwall_1;

       // Bit 5
       "DB_PLC_ISO_IHM".Cleaning_Backwall_2 := "DB_PLC_ISO_IHM".Cleaning_Backwall_2;

       // Bit 6
       "DB_PLC_ISO_IHM".Shutter_laser_closed := "DB_DigitalInputs".sShutterClosed.sSWStatus OR
            NOT "DB_DataFromSafety".iKeyLaserOn;

       // Bit 7
       "DB_PLC_ISO_IHM".Pressure_Stop_Machine := "DB_PLC_ISO_IHM".Pressure_Stop_Machine;
   END_REGION

   REGION Byte 971  
       // Bit 0
       IF "LBP_Chan1".MDyn[68] OR "DB_Scanner".sScannerComm.oGoodPart THEN
           "DB_PLC_ISO_IHM".BadPartOnFixture := FALSE;
       ELSIF "DB_BadPartOnFixture".BadPartOnFixture
           OR "DB_GestionFixture".sFixturePartControl.oBadpart
           OR "DB_Scanner".sScannerComm.oBadPart THEN
               "DB_PLC_ISO_IHM".BadPartOnFixture := TRUE;
       END_IF;

       // Bit 1 (NOT USED ON FL0125)
       "DB_PLC_ISO_IHM".Reserve12 := "DB_PLC_ISO_IHM".Reserve12;

       // Bit 2 (NOT USED ON FL0125)
       "DB_PLC_ISO_IHM".Reserve13 := "DB_PLC_ISO_IHM".Reserve13;

       // Bit 3 (NOT USED ON FL0125)
       "DB_PLC_ISO_IHM".Reserve14 := "DB_PLC_ISO_IHM".Reserve14;

       // Bit 4 (NOT USED ON FL0125)
       "DB_PLC_ISO_IHM".Reserve15 := "DB_PLC_ISO_IHM".Reserve15;

       // Bit 5
       "DB_PLC_ISO_IHM".SemiAuto_RunEmpty := "DB_PLC_ISO_IHM".SemiAuto_RunEmpty;

       // Bit 6
       "DB_PLC_ISO_IHM"."SemiAuto_Unload_C-Fixture" := "DB_PLC_ISO_IHM"."SemiAuto_Unload_C-Fixture";

       // Bit 7 (NOT USED ON FL0125)
       "DB_PLC_ISO_IHM".Reserve18 := "DB_PLC_ISO_IHM".Reserve18;
   END_REGION

   REGION Transfert data PLC -> ISO

       FOR #tLoop := 0 TO 11 DO
           #sTransferActData[#tLoop] := PEEK(area := 16#84, dbNumber := 1302, byteOffset := #tLoop);
           IF #sTransferActData[#tLoop] <> #sTransferSelData[#tLoop] THEN
               #sUpdate_PLC_ISO_Values := TRUE;
               #sTransferSelData[#tLoop] := #sTransferActData[#tLoop];
           END_IF;
       END_FOR;

       // Transfert DB_PLC_ISO_IHM DWORD 0  

       // DEFINE PART_ON_FIXTURE_1         AS (($A_DBB[963] B_AND 1)==1)
       // DEFINE MASTER_ON_FIXTURE_1       AS (($A_DBB[963] B_AND 2)==2)
       // DEFINE CAN_CHANGE_PART_LOADER_2  AS (($A_DBB[963] B_AND 4)==4)
       // DEFINE CHECK_PART_FIXTURE_2      AS (($A_DBB[963] B_AND 8)==8)
       // DEFINE LOADER_2_PART_LOAD        AS (($A_DBB[963] B_AND 16)==16)
       // DEFINE LOADER_2_PART_UNLOAD      AS (($A_DBB[963] B_AND 32)==32)
       // DEFINE LOADER_2_SHIFT_LOAD       AS (($A_DBB[963] B_AND 64)==64)
       // DEFINE LOADER_2_SHIFT_UNLOAD     AS (($A_DBB[963] B_AND 128)==128)

       "LBP_TransferSelData"(Enable := #sUpdate_PLC_ISO_Values,
                             Funct := BYTE#16#04,
                             IVAR1 := 963,
                             IVAR2 := -1,
                             Error => #tTransferSelDataError.%X0,
                             ErrCode => #tTransferSelDataErrCode[0],
                             S7Var := #sTransferSelData[3]);

       // DEFINE CAN_CHANGE_PART_LOADER_1  AS (($A_DBB[962] B_AND 1)==1)
       // DEFINE CHECK_PART_FIXTURE_1      AS (($A_DBB[962] B_AND 2)==2)
       // DEFINE LOADER_1_PART_LOAD        AS (($A_DBB[962] B_AND 4)==4)
       // DEFINE LOADER_1_PART_UNLOAD      AS (($A_DBB[962] B_AND 8)==8)
       // DEFINE LOADER_1_SHIFT_LOAD       AS (($A_DBB[962] B_AND 16)==16)
       // DEFINE LOADER_1_SHIFT_UNLOAD     AS (($A_DBB[962] B_AND 32)==32)
       // DEFINE LOADER_1_LOAD_OPENED      AS (($A_DBB[962] B_AND 64)==64)
       // DEFINE LOADER_1_UNLOAD_OPENED    AS (($A_DBB[962] B_AND 128)==128)

       "LBP_TransferSelData"(Enable := #sUpdate_PLC_ISO_Values,
                             Funct := BYTE#16#04,
                             IVAR1 := 962,
                             IVAR2 := -1,
                             Error => #tTransferSelDataError.%X1,
                             ErrCode => #tTransferSelDataErrCode[1],
                             S7Var := #sTransferSelData[2]);

       // DEFINE STOP_AT_NEXT_REQ          AS (($A_DBB[961] B_AND 1)==1)
       // DEFINE ALL_CHAN_STOP             AS (($A_DBB[961] B_AND 2)==2)
       // DEFINE LOADER_MODE_AUTOMATIC     AS (($A_DBB[961] B_AND 4)==4)
       // DEFINE LOADER_MODE_MANUAL        AS (($A_DBB[961] B_AND 8)==8)
       // DEFINE MODE_WITH_LOADER          AS (($A_DBB[961] B_AND 12)>0)
       // DEFINE MODE_WITHOUT_LOADER       AS (($A_DBB[961] B_AND 12)==0)
       // DEFINE NO_CAMERA_PRESENT         AS (($A_DBB[961] B_AND 16)==16)
       // DEFINE PREMEASURE_Z_EXISTS       AS (($A_DBB[961] B_AND 32)==32)
       // DEFINE PREMEASURE_C_EXISTS       AS (($A_DBB[961] B_AND 64)==64)

       "LBP_TransferSelData"(Enable := #sUpdate_PLC_ISO_Values,
                             Funct := BYTE#16#04,
                             IVAR1 := 961,
                             IVAR2 := -1,
                             Error => #tTransferSelDataError.%X2,
                             ErrCode => #tTransferSelDataErrCode[2],
                             S7Var := #sTransferSelData[1]);

       // DEFINE WARM_UP_ON                AS (($A_DBB[960] B_AND 1)==1)
       // DEFINE KEY_LASER_ON              AS (($A_DBB[960] B_AND 2)==2)
       // DEFINE KEY_SAVE_PARAM            AS (($A_DBB[960] B_AND 4)==4)
       // DEFINE STOP_PROG_RUN             AS (($A_DBB[960] B_AND 8)==8)
       // DEFINE CHAN_1_RUNNING            AS (($A_DBB[960] B_AND 16)==16)
       // DEFINE CHAN_2_RUNNING            AS (($A_DBB[960] B_AND 32)==32)
       // DEFINE CHAN_3_RUNNING            AS (($A_DBB[960] B_AND 64)==64)
       // DEFINE CHAN_4_RUNNING            AS (($A_DBB[960] B_AND 128)==128)

       "LBP_TransferSelData"(Enable := #sUpdate_PLC_ISO_Values,
                             Funct := BYTE#16#04,
                             IVAR1 := 960,
                             IVAR2 := -1,
                             Error => #tTransferSelDataError.%X3,
                             ErrCode => #tTransferSelDataErrCode[3],
                             S7Var := #sTransferSelData[0]);

       // Transfert DB_PLC_ISO_IHM DWORD 4  


       "LBP_TransferSelData"(Enable := #sUpdate_PLC_ISO_Values,
                             Funct := BYTE#16#04,
                             IVAR1 := 967,
                             IVAR2 := -1,
                             Error => #tTransferSelDataError.%X4,
                             ErrCode => #tTransferSelDataErrCode[4],
                             S7Var := #sTransferSelData[7]);

       "LBP_TransferSelData"(Enable := #sUpdate_PLC_ISO_Values,
                             Funct := BYTE#16#04,
                             IVAR1 := 966,
                             IVAR2 := -1,
                             Error => #tTransferSelDataError.%X5,
                             ErrCode => #tTransferSelDataErrCode[5],
                             S7Var := #sTransferSelData[6]);

       // DEFINE LOADER_3_SHIFT_LOAD       AS (($A_DBB[965] B_AND 1)==1)
       // DEFINE LOADER_3_SHIFT_UNLOAD     AS (($A_DBB[965] B_AND 2)==2)
       // DEFINE LOADER_3_LOAD_OPENED      AS (($A_DBB[965] B_AND 4)==4)
       // DEFINE LOADER_3_UNLOAD_OPENED    AS (($A_DBB[965] B_AND 8)==8)
       // DEFINE PART_ON_FIXTURE_3         AS (($A_DBB[965] B_AND 16)==16)
       // DEFINE MASTER_ON_FIXTURE_3       AS (($A_DBB[965] B_AND 32)==32)
       // DEFINE PART_KO_GO_OUTSIDE        AS (($A_DBB[965] B_AND 64)==64)
       // DEFINE MASTER_ON_MACHINE         AS (($A_DBB[965] B_AND 128)==128)

       "LBP_TransferSelData"(Enable := #sUpdate_PLC_ISO_Values,
                             Funct := BYTE#16#04,
                             IVAR1 := 965,
                             IVAR2 := -1,
                             Error => #tTransferSelDataError.%X6,
                             ErrCode => #tTransferSelDataErrCode[6],
                             S7Var := #sTransferSelData[5]);

       // DEFINE LOADER_2_LOAD_OPENED      AS (($A_DBB[964] B_AND 1)==1)
       // DEFINE LOADER_2_UNLOAD_OPENED    AS (($A_DBB[964] B_AND 2)==2)
       // DEFINE PART_ON_FIXTURE_2         AS (($A_DBB[964] B_AND 4)==4)
       // DEFINE MASTER_ON_FIXTURE_2       AS (($A_DBB[964] B_AND 8)==8)
       // DEFINE CAN_CHANGE_PART_LOADER_3  AS (($A_DBB[964] B_AND 16)==16)
       // DEFINE CHECK_PART_FIXTURE_3      AS (($A_DBB[964] B_AND 32)==32)
       // DEFINE LOADER_3_PART_LOAD        AS (($A_DBB[964] B_AND 64)==64)
       // DEFINE LOADER_3_PART_UNLOAD      AS (($A_DBB[964] B_AND 128)==128)

       "LBP_TransferSelData"(Enable := #sUpdate_PLC_ISO_Values,
                             Funct := BYTE#16#04,
                             IVAR1 := 964,
                             IVAR2 := -1,
                             Error => #tTransferSelDataError.%X7,
                             ErrCode => #tTransferSelDataErrCode[7],
                             S7Var := #sTransferSelData[4]);

       // Transfert DB_PLC_ISO_IHM DWORD 8  

       // DEFINE SET_BAD_PART_ON_FIXTURE   AS (($A_DBB[971] B_AND 1)==1)
       // ;DEFINE     AS (($A_DBB[971] B_AND 2)==2)
       // ;DEFINE     AS (($A_DBB[971] B_AND 4)==4)
       // ;DEFINE     AS (($A_DBB[971] B_AND 8)==8)
       // ;DEFINE     AS (($A_DBB[971] B_AND 16)==16)
       // DEFINE SEMIAUTO_RUNEMPTY         AS (($A_DBB[971] B_AND 32)==32)
       // DEFINE SEMIAUTO_UNLOAD_C_FIXTURE AS (($A_DBB[971] B_AND 64)==64)
       // ;DEFINE     AS (($A_DBB[971] B_AND 128)==128

       "LBP_TransferSelData"(Enable := #sUpdate_PLC_ISO_Values,
                             Funct := BYTE#16#04,
                             IVAR1 := 971,
                             IVAR2 := -1,
                             Error => #tTransferSelDataError.%X8,
                             ErrCode => #tTransferSelDataErrCode[8],
                             S7Var := #sTransferSelData[11]);

       // DEFINE STOP_FOR_BACKWALL1_WEARED AS (($A_DBB[970] B_AND 1)==1)
       // DEFINE STOP_FOR_BACKWALL2_WEARED AS (($A_DBB[970] B_AND 2)==2)
       // DEFINE CLEANING_STATION1         AS (($A_DBB[970] B_AND 4)==4)
       // DEFINE CLEANING_STATION2         AS (($A_DBB[970] B_AND 8)==8)
       // DEFINE CLEANING_BACKWALL1        AS (($A_DBB[970] B_AND 16)==16)
       // DEFINE CLEANING_BACKWALL2        AS (($A_DBB[970] B_AND 32)==32)
       // DEFINE LASER_SHUTTER_CLOSED      AS (($A_DBB[970] B_AND 64)==64)
       // DEFINE NOT_COND_FOR_DRILL        AS (($A_DBB[970] B_AND 128)==128)

       "LBP_TransferSelData"(Enable := #sUpdate_PLC_ISO_Values,
                             Funct := BYTE#16#04,
                             IVAR1 := 970,
                             IVAR2 := -1,
                             Error => #tTransferSelDataError.%X9,
                             ErrCode => #tTransferSelDataErrCode[9],
                             S7Var := #sTransferSelData[10]);


       "LBP_TransferSelData"(Enable := #sUpdate_PLC_ISO_Values,
                             Funct := BYTE#16#04,
                             IVAR1 := 969,
                             IVAR2 := -1,
                             Error => #tTransferSelDataError.%X10,
                             ErrCode => #tTransferSelDataErrCode[10],
                             S7Var := #sTransferSelData[9]);

       // DEFINE WARM_UP_TIME              AS ($A_DBW[968])

       "LBP_TransferSelData"(Enable := #sUpdate_PLC_ISO_Values,
                             Funct := BYTE#16#04,
                             IVAR1 := 968,
                             IVAR2 := -1,
                             Error => #tTransferSelDataError.%X11,
                             ErrCode => #tTransferSelDataErrCode[11],
                             S7Var := #sTransferSelData[8]);

       IF #tTransferSelDataError = 0 THEN
           #sUpdate_PLC_ISO_Values := FALSE;
       END_IF;
   END_REGION
END_FUNCTION_BLOCK

FUNCTION_BLOCK "FB_Alarms_Safety"   // FB150, SCL
{ S7_Optimized_Access := 'TRUE' }
// stored: AutoNumber false, MemoryReserve 100, SetENOAutomatically false
   VAR
      sTimerEmergencyPowLaser : IEC_TIMER;
   END_VAR
BEGIN
   REGION Description header 
       //==================================================================================
       // POSALUX Swiss SA / (C) Copyright 2024
       //----------------------------------------------------------------------------------
       // Title: Affichage Alarmes/Messages Safety
       // Comment/Function: 
       //
       // Author: Michel FAIVRE
       // Engineering: TIA Portal v17
       //----------------------------------------------------------------------------------
       // Change log table:
       // Version  | Date     | Expert in charge | Changes applied
       // ---------|----------|------------------|------------------------------------
       // 01.01.00 | 20241218 | FMI              | First released version
       // ==================================================================================
   END_REGION

   REGION Warnings
       // Warning 700236 : Shutter ready to open, press laser button
       IF "LBP_AlarmMsgs".UserA[2].A70UUxx[36] AND
           ("MCP1_In".reset OR "DB_DataFromSafety".OpenShutter) THEN
           "LBP_AlarmMsgs".UserA[2].A70UUxx[36] := False;
       END_IF;
       IF NOT "LBP_AlarmMsgs".UserA[2].A70UUxx[36] AND NOT "DB_DataFromSafety".OpenShutter AND
           "DB_PowerOn".sMachinePower AND
           "DB_DataFromSafety".EmergencyStop AND
           "DB_DataFromSafety".iEmergencyStopPowerLaser AND
           "DB_DataFromSafety".iKeyLaserOn AND
           ("DB_DataFromSafety".iKeySettingLaser OR "DB_DataFromSafety".AllDoorLockedForLaser) THEN
           "LBP_AlarmMsgs".UserA[2].A70UUxx[36] := True;
       END_IF;

       // Warnings Doors
       "LBP_AlarmMsgs".UserA[5].A70UUxx[37] := NOT "DB_DataFromSafety".iFrontDoorClosed;
       "LBP_AlarmMsgs".UserA[5].A70UUxx[38] := NOT "DB_DataFromSafety".iMaintenanceDoorClosed;
       "LBP_AlarmMsgs".UserA[5].A70UUxx[39] := NOT "DB_DataFromSafety".iRoofLeftDoorClosed;
       "LBP_AlarmMsgs".UserA[5].A70UUxx[48] := NOT "DB_DataFromSafety".iRoofRightDoorClosed;

       // Warning 700542 : SAFETY : FEED STOP FOR ALL AXIS, MAIN DOOR IS CLOSED BUT NOT LOCKED
       IF "DB_DataFromSafety".iFrontDoorClosed
           AND NOT "DB_DigitalInputs".sFrontDoorLocked.sSWStatus  // Control Front Door locked
           AND "DB_DataFromSafety".iRoofLeftDoorClosed
           AND "DB_DataFromSafety".iRoofRightDoorClosed
           AND "DB_DataFromSafety".iKeySettingMode
           AND NOT "DB_McpKeyboardSignals".sAlarmReset.sKeySWStatus THEN
           IF "MCP1_In".minus OR "MCP1_In".plus THEN
               "LBP_AlarmMsgs".UserA[5].A70UUxx[42] := TRUE;
           END_IF;
       ELSE
           "LBP_AlarmMsgs".UserA[5].A70UUxx[42] := FALSE;
       END_IF;

       // Warning 700532 : SAFETY : COMMISSIONNING ON
       "LBP_AlarmMsgs".UserA[5].A70UUxx[32] := "DB_DataFromSafety".Comissionning;

       // Warning 700533 : SAFETY : LASER POWER SUPPLY IN EMERGENCY STOP
       #sTimerEmergencyPowLaser.TON(PT := t#200ms,
                                    IN := NOT "DB_DataFromSafety".iEmergencyStopPowerLaser);
       "LBP_AlarmMsgs".UserA[5].A70UUxx[33] := #sTimerEmergencyPowLaser.Q;

       // Warning 700534 : SAFETY : LASER SETTING MODE IS ACTIVE
       "LBP_AlarmMsgs".UserA[5].A70UUxx[34] := "DB_DataFromSafety".iKeySettingLaser;

       // Warning 700535 : SAFETY : LASER SHUTTER IS CLOSED
       "LBP_AlarmMsgs".UserA[5].A70UUxx[35] := "DB_DataFromSafety".ShutterClosed;

       // Warning 700536 : SAFETY : FEED STOP FOR ALL AXIS, PLEASE TURN SETTING KEY TO MOVE AXIS
       "LBP_AlarmMsgs".UserA[5].A70UUxx[36] := NOT "DB_DataFromSafety".DoorsClosed AND NOT "DB_DataFromSafety".iKeySettingMode;

       // Warning 700550 : SAFETY : KEY LASER OFF
       "LBP_AlarmMsgs".UserA[5].A70UUxx[50] := NOT "DB_DataFromSafety".iKeyLaserOn;

       // Warning 700551 : SAFETY : KEY LASER ON BUT LASER NOT READY
       "LBP_AlarmMsgs".UserA[5].A70UUxx[51] := "DB_DataFromSafety".iKeyLaserOn
       AND NOT "DB_DataFromSafety".ShutterReadyToOpen;

       // Warning 700552 : SAFETY : KEY LASER ON, LASER READY, SHUTTER CLOSED BY SOURCE
       // A implementer si l'entrée I0.7 SHUTTER IS CLOSED existe
       // "LBP_AlarmMsgs".UserA[5].A70UUxx[52] := "Main_Safety_RTG1_DB".SAFETY_LASER_KEY_ON
       // AND "Main_Safety_RTG1_DB".sLaserSupplyPower
       // AND "Main_Safety_RTG1_DB".SAFETY_EMERGENCY_STOP_POWER_LASER
       // AND (Shutter_is_closed) ;


   END_REGION

   REGION Alarms
       // Alarm 700500 : SAFETY : EMERGENCY STOP IS ACTIVE, PLEASE RESET  
       IF "DB_DataFromSafety".AckEmergencyStop THEN
           "LBP_AlarmMsgs".UserA[5].A70UUxx[0] := TRUE;
       END_IF;
       //  "LBP_AlarmMsgs".UserA[5].A70UUxx[0] := "DB_DataFromSafety".AckEmergencyStop;

       // Alarm 700501 : SAFETY : LASER POWER SUPPLY IS OFF, PLEASE RESET  
       IF NOT "DB_DataFromSafety".oContactorLaser THEN
           "LBP_AlarmMsgs".UserA[5].A70UUxx[1] := TRUE;
       END_IF;
       //   "LBP_AlarmMsgs".UserA[5].A70UUxx[1] := NOT "DB_DataFromSafety".oContactorLaser;

       // Alarm 700502 :SAFETY : LASER POWER SUPPLY IS NOT READY , PLEASE RESET
       IF NOT "DB_DataFromSafety".iEmergencyStopPowerLaser
           AND "DB_CycleStartStop".sChan1Start THEN
           "LBP_AlarmMsgs".UserA[5].A70UUxx[2] := TRUE;
       END_IF;

       // Alarm 700508 : SAFETY : FEEDBACK CONTACTOR POWER MACHINE IS NOT WORKING , PLEASE RESET
       IF "DB_DataFromSafety".SupplyPowerError AND "DB_PowerOn".sMachineReadySoft THEN
           "LBP_AlarmMsgs".UserA[5].A70UUxx[8] := TRUE;
       END_IF;

       // Alarm 700509 : SAFETY : FEEDBACK CONTACTOR POWER LASER IS NOT WORKING , PLEASE RESET
       IF "DB_DataFromSafety".LaserSupplyPowerError THEN
           "LBP_AlarmMsgs".UserA[5].A70UUxx[9] := TRUE;
       END_IF;

       // Alarm 700510 : SAFETY : FEEDBACK CONTACTOR OPEN SHUTTER IS NOT WORKING , PLEASE RESET
       IF "DB_DataFromSafety".ShutterError THEN
           "LBP_AlarmMsgs".UserA[5].A70UUxx[10] := TRUE;
       END_IF;

       // Alarm 700511 : SAFETY : FATAL ERROR ! : WRONG DISCORDANCE BEETWEEN SAFETY INPUTS, PLEASE RESET AND CHANGE SETTINGS
       "LBP_AlarmMsgs".UserA[5].A70UUxx[11] := "DB_DataFromSafety".AckI2001Functions;
   END_REGION
END_FUNCTION_BLOCK

FUNCTION_BLOCK "FB_LoaderMain"   // FB203, SCL
{ S7_Optimized_Access := 'TRUE' }
// stored: AutoNumber false, MemoryReserve 100, SetENOAutomatically false
   VAR
      sSynchroMode : Bool;
      sSynchroPosition : Bool;
      sLoaderStartRequest : Bool;
      sTimeMeasure : "FB_TimeMeasure";
      sRT_LoaderStartRequest { S7_SetPoint := 'True'} : R_TRIG;
      sBwConsecutiveCtrl { S7_SetPoint := 'True'} : "FB_Consecutive";
      sRT_ConsecutiveCtrl { S7_SetPoint := 'True'} : R_TRIG;
   END_VAR
BEGIN
   REGION Description header 
       //==================================================================================
       // POSALUX Swiss SA / (C) Copyright 2025
       //----------------------------------------------------------------------------------
       // Title: 
       // Comment/Function: 
       // Author: Fabien WALDT
       // Engineering: TIA Portal v17
       //----------------------------------------------------------------------------------
       // Change log table:
       // Version  | Date     | Expert in charge | Changes applied
       // ---------|----------|------------------|-----------------------------------------
       // 00.00.01 | 20251013 | WFA              | First released version
       // =================================================================================
   END_REGION

   REGION Options
       // Ext Load Unload
       "DB_LoaderOptions".ExtLoadUnload.SeparatePos := FALSE;
       "DB_LoaderOptions".ExtLoadUnload.CommonPos := TRUE;
       // Part Control
       "DB_LoaderOptions".PartControl.Individual := FALSE;
       "DB_LoaderOptions".PartControl.Common := TRUE;
       "DB_LoaderOptions".PartControl.Disabled := FALSE;
       "DB_LoaderOptions".PartControl.AnalogMeasure := FALSE;
       "DB_LoaderOptions".PartControl.DigitalMeasure := TRUE;
       // BW Load Unload
       "DB_LoaderOptions".BwLoadUnload.SeparatePos := TRUE;
       "DB_LoaderOptions".BwLoadUnload.CommonPos := FALSE;
       // BW Control
       "DB_LoaderOptions".BwControl.UndrilledDrilledCtrlSeparate := TRUE;
       "DB_LoaderOptions".BwControl.UndrilledDrilledCtrlCommon := FALSE;
       "DB_LoaderOptions".BwControl.Disabled := FALSE;
       // Int Load Unload
       "DB_LoaderOptions".IntLoadUnload.SeparatePos := FALSE;
       "DB_LoaderOptions".IntLoadUnload.CommonPos := TRUE;
   END_REGION

   REGION History Activation
       // Shuttle 1
       "DB_LoaderShuttle1".sMain.sHistory.Activation := TRUE;
       "DB_LoaderShuttle1".sShuttleInt.sHistory.Activation := TRUE;
       "DB_LoaderShuttle1".sShuttleExt.sHistory.Activation := TRUE;
       "DB_LoaderShuttle1".sControlIn.sHistory.Activation := TRUE;
       "DB_LoaderShuttle1".sControlOut.sHistory.Activation := TRUE;
       "DB_LoaderShuttle1".sIntLoadUnload.sHistory.Activation := TRUE;
       "DB_LoaderShuttle1".sIntLoadUnloadOP.sHistory.Activation := TRUE;
       "DB_LoaderShuttle1".sExtLoadUnload.sHistory.Activation := TRUE;
       "DB_LoaderShuttle1".sBwLoadUnload.sHistory.Activation := TRUE;
       "DB_LoaderShuttle1".sBwControlIn.sHistory.Activation := TRUE;
       "DB_LoaderShuttle1".sActBwControlIn.sHistory.Activation := TRUE;
       "DB_LoaderShuttle1".sActPartControlIn.sHistory.Activation := TRUE;
       "DB_LoaderShuttle1".sActPartControlOut.sHistory.Activation := TRUE;
       "DB_LoaderShuttle1".sBlowing.sHistory.Activation := TRUE;

       // Shuttle 2
       "DB_LoaderShuttle2".sMain.sHistory.Activation := TRUE;
       "DB_LoaderShuttle2".sShuttleInt.sHistory.Activation := TRUE;
       "DB_LoaderShuttle2".sShuttleExt.sHistory.Activation := TRUE;
       "DB_LoaderShuttle2".sControlIn.sHistory.Activation := TRUE;
       "DB_LoaderShuttle2".sControlOut.sHistory.Activation := TRUE;
       "DB_LoaderShuttle2".sIntLoadUnload.sHistory.Activation := TRUE;
       "DB_LoaderShuttle2".sIntLoadUnloadOP.sHistory.Activation := TRUE;
       "DB_LoaderShuttle2".sExtLoadUnload.sHistory.Activation := TRUE;
       "DB_LoaderShuttle2".sBwLoadUnload.sHistory.Activation := TRUE;
       "DB_LoaderShuttle2".sBwControlIn.sHistory.Activation := TRUE;
       "DB_LoaderShuttle2".sActBwControlIn.sHistory.Activation := TRUE;
       "DB_LoaderShuttle2".sActPartControlIn.sHistory.Activation := TRUE;
       "DB_LoaderShuttle2".sActPartControlout.sHistory.Activation := TRUE;
       "DB_LoaderShuttle2".sBlowing.sHistory.Activation := TRUE;
   END_REGION

   REGION Loader Start
       IF "LBP_Chan1".MDyn[75] AND ("DB_WorkingModes".sAuto OR "DB_WorkingModes".sSemiAuto) THEN
           #sLoaderStartRequest := TRUE;
       ELSIF
           ("DB_WorkingModes".sEmptying AND "DB_PartManagement".sPosition.sMachineEmpty)
          OR NOT "DB_PowerOn".sMachineReadySoft
          OR  "MCP1_In".reset THEN
           #sLoaderStartRequest := FALSE;
       END_IF;

           #sRT_LoaderStartRequest(CLK := #sLoaderStartRequest);
           IF NOT "LBP_ModeGroup".E_JOG AND #sRT_LoaderStartRequest.Q THEN
               IF "DB_HMISetting".Shuttle1Enable THEN
                   "DB_LoaderShuttle1".sMain.iJobReq := TRUE;
               END_IF;
               IF "DB_HMISetting".Shuttle2Enable THEN
                   "DB_LoaderShuttle2".sMain.iJobReq := TRUE;
               END_IF;
           ELSIF NOT #sLoaderStartRequest THEN
               "DB_LoaderShuttle1".sMain.iJobReq := FALSE;
               "DB_LoaderShuttle2".sMain.iJobReq := FALSE;
           END_IF;
   END_REGION

   REGION Shuttle 1
       "DB_LoaderShuttle1"(iGripperReserved := "DB_GestionGripper".sGripperStatus.DrivedByShuttle1,
                           iGripperReleased := NOT "DB_GestionGripper".sGripperStatus.DrivedByShuttle1,
                           iShuttleMoving := "DB_LoaderAxis".sU1Positioning,
                           iShuttleInPos := "DB_LoaderAxis".sU1InPos,
                           iAxisV_Moving := "DB_LoaderAxis".sVPositioning,
                           iAxisV_InPos := "DB_LoaderAxis".sVInPos,
                           iAxisW_Moving := "DB_LoaderAxis".sWPositioning,
                           iAxisW_InPos := "DB_LoaderAxis".sWInPos,
                           oExtGateOpenReq => "DB_LoaderShuttle1".oExtGateOpenReq,
                           oExtGateCloseReq => "DB_LoaderShuttle1".oExtGateCloseReq,
                           oIntGateOpenReq => "DB_LoaderShuttle1".oIntGateOpenReq,
                           oIntGateCloseReq => "DB_LoaderShuttle1".oIntGateCloseReq,
                           oLoadGripperCloseReq => "DB_LoaderShuttle1".oLoadGripperCloseReq,
                           oUnloadGripperOpenReq => "DB_LoaderShuttle1".oUnloadGripperOpenReq,
                           oShuttleStartReq => "DB_LoaderShuttle1".oShuttleStartReq,
                           oShuttlePosSetPoint => "DB_LoaderAxis".iU1PosSetPoint,
                           oAxisVStartReq => "DB_LoaderShuttle1".oAxisVStartReq,
                           oAxisVPosSetPoint => "DB_LoaderShuttle1".oAxisVPosSetPoint,
                           oAxisWStartReq => "DB_LoaderShuttle1".oAxisWStartReq,
                           oAxisWPosSetPoint => "DB_LoaderShuttle1".oAxisWPosSetPoint);
   END_REGION

   REGION Shuttle 2
       "DB_LoaderShuttle2"(iGripperReserved := "DB_GestionGripper".sGripperStatus.DrivedByShuttle2,
                           iGripperReleased :=  NOT "DB_GestionGripper".sGripperStatus.DrivedByShuttle2,
                           iShuttleMoving := "DB_LoaderAxis".sU2Positioning,
                           iShuttleInPos := "DB_LoaderAxis".sU2InPos,
                           iAxisV_Moving := "DB_LoaderAxis".sVPositioning,
                           iAxisV_InPos := "DB_LoaderAxis".sVInPos,
                           iAxisW_Moving := "DB_LoaderAxis".sWPositioning,
                           iAxisW_InPos := "DB_LoaderAxis".sWInPos,
                           oExtGateOpenReq => "DB_LoaderShuttle2".oExtGateOpenReq,
                           oExtGateCloseReq => "DB_LoaderShuttle2".oExtGateCloseReq,
                           oIntGateOpenReq => "DB_LoaderShuttle2".oIntGateOpenReq,
                           oIntGateCloseReq => "DB_LoaderShuttle2".oIntGateCloseReq,
                           oLoadGripperCloseReq => "DB_LoaderShuttle2".oLoadGripperCloseReq,
                           oUnloadGripperOpenReq => "DB_LoaderShuttle2".oUnloadGripperOpenReq,
                           oShuttleStartReq => "DB_LoaderShuttle2".oShuttleStartReq,
                           oShuttlePosSetPoint => "DB_LoaderAxis".iU2PosSetPoint,
                           oAxisVStartReq => "DB_LoaderShuttle2".oAxisVStartReq,
                           oAxisVPosSetPoint => "DB_LoaderShuttle2".oAxisVPosSetPoint,
                           oAxisWStartReq => "DB_LoaderShuttle2".oAxisWStartReq,
                           oAxisWPosSetPoint => "DB_LoaderShuttle2".oAxisWPosSetPoint);
   END_REGION

   REGION Loader Axis
       IF "DB_LoaderShuttle1".oAxisVStartReq THEN
           "DB_LoaderAxis".iVPosSetPoint := "DB_LoaderShuttle1".oAxisVPosSetPoint;
       ELSIF "DB_LoaderShuttle2".oAxisVStartReq THEN
           "DB_LoaderAxis".iVPosSetPoint := "DB_LoaderShuttle2".oAxisVPosSetPoint;
       ELSIF "DB_LoaderFixture".oAxisV_StartReq THEN
           "DB_LoaderAxis".iVPosSetPoint := "DB_LoaderFixture".oAxisV_PosSetPoint;
       END_IF;

       IF "DB_LoaderShuttle1".oAxisWStartReq THEN
           "DB_LoaderAxis".iWPosSetPoint := "DB_LoaderShuttle1".oAxisWPosSetPoint;
       ELSIF "DB_LoaderShuttle2".oAxisWStartReq THEN
           "DB_LoaderAxis".iWPosSetPoint := "DB_LoaderShuttle2".oAxisWPosSetPoint;
       ELSIF "DB_LoaderFixture".oAxisW_StartReq THEN
           "DB_LoaderAxis".iWPosSetPoint := "DB_LoaderFixture".oAxisW_PosSetPoint;
       END_IF;

       // Demande Axes gérés par PLC (/Mode Jog)
       IF "LBP_ModeGroup".E_MDA OR "LBP_ModeGroup".E_AUTO THEN
           "DB_LoaderAxis".iPLCModeReq := TRUE;
       ELSE
           "DB_LoaderAxis".iPLCModeReq := FALSE;
       END_IF;

       // Demande Axes gérés par NC (Mode Jog)
       // Jog Mode OR R_Trig Auto Mode
           IF "LBP_ModeGroup".E_JOG  THEN
           "DB_LoaderAxis".iCNCModeReq := TRUE;
       ELSE
           "DB_LoaderAxis".iCNCModeReq := FALSE;
       END_IF;

       "DB_LoaderAxis"(iPLCModeReq := "DB_LoaderAxis".iPLCModeReq,
                       iCNCModeReq := "DB_LoaderAxis".iCNCModeReq,
                       iU1StartReq := "DB_LoaderShuttle1".oShuttleStartReq,
                       iU2StartReq := "DB_LoaderShuttle2".oShuttleStartReq,
                       iVStartReq := "DB_LoaderShuttle1".oAxisVStartReq OR "DB_LoaderShuttle2".oAxisVStartReq OR "DB_LoaderFixture".oAxisV_StartReq,
                       iWStartReq := "DB_LoaderShuttle1".oAxisWStartReq OR "DB_LoaderShuttle2".oAxisWStartReq OR "DB_LoaderFixture".oAxisW_StartReq,
                       iU1PosSetPoint := "DB_LoaderAxis".iU1PosSetPoint,
                       iU2PosSetPoint := "DB_LoaderAxis".iU2PosSetPoint,
                       iVPosSetPoint := "DB_LoaderAxis".iVPosSetPoint,
                       iWPosSetPoint := "DB_LoaderAxis".iWPosSetPoint,
                       oU1InPos => "DB_LoaderAxis".oU1InPos,
                       oU2InPos => "DB_LoaderAxis".oU2InPos,
                       oVInPos => "DB_LoaderAxis".oVInPos,
                       oWInPos => "DB_LoaderAxis".oWInPos);
   END_REGION

   REGION Safety Gate
       "DB_GestionSafetyGate"();
   END_REGION

   REGION Gripper
       "DB_GestionGripper"();
   END_REGION

   REGION Fixture
       "DB_GestionFixture"();
   END_REGION

   REGION Syncro Mode 
       // WFA Tester le cycle en supprimant cette REGION (voir tSynchroMode dans FB_GestionSafetyGate)
       #sSynchroMode := "DB_LoaderShuttle1".sMain.sInterface.SequenceRun
       AND "DB_LoaderShuttle2".sMain.sInterface.SequenceRun
       AND (("DB_LoaderShuttle1".sShuttleInt.oExtGateOpenReq AND "DB_LoaderShuttle2".sShuttlePosSas)
       OR ("DB_LoaderShuttle1".sShuttleInt.oIntGateOpenReq AND "DB_LoaderShuttle2".sShuttlePosInt)
       OR ("DB_LoaderShuttle1".sShuttleExt.oExtGateOpenReq AND "DB_LoaderShuttle2".sShuttlePosExt)
       OR ("DB_LoaderShuttle1".sShuttleExt.oIntGateOpenReq AND "DB_LoaderShuttle2".sShuttlePosSas)
       OR ("DB_LoaderShuttle2".sShuttleInt.oExtGateOpenReq AND "DB_LoaderShuttle1".sShuttlePosSas)
       OR ("DB_LoaderShuttle2".sShuttleInt.oIntGateOpenReq AND "DB_LoaderShuttle1".sShuttlePosInt)
       OR ("DB_LoaderShuttle2".sShuttleExt.oExtGateOpenReq AND "DB_LoaderShuttle1".sShuttlePosExt)
       OR ("DB_LoaderShuttle2".sShuttleExt.oIntGateOpenReq AND "DB_LoaderShuttle1".sShuttlePosSas));
   END_REGION

   REGION Time Measure
       #sTimeMeasure(iImpulsion := "DB_GestionGripper".sLoadGripperCloseReq,
                     iPLC_DateAndTime := "DB_ReadDateAndTime".sDateAndTime);
   END_REGION

   REGION Consecutive
       IF "DB_OPC_Machine".Parameters.ConsecutiveBwIn > 0 THEN
           #sBwConsecutiveCtrl(iReset := #sBwConsecutiveCtrl.oConsecutiveError AND ("DB_McpKeyboardSignals".sAlarmReset.sKeySWStatus OR "MCP1_In".reset),
                               iGoodEntry := "DB_LoaderShuttle1".sBwControlIn.oBwControlOK OR "DB_LoaderShuttle2".sBwControlIn.oBwControlOK,
                               iBadEntry := "DB_LoaderShuttle1".sBwControlIn.oBwControlNOK OR "DB_LoaderShuttle2".sBwControlIn.oBwControlNOK,
                               iPresetValue := "DB_OPC_Machine".Parameters.ConsecutiveBwIn,
                               oConsecutiveError => #sBwConsecutiveCtrl.oConsecutiveError);

           #sRT_ConsecutiveCtrl(CLK := #sBwConsecutiveCtrl.oConsecutiveError);
           IF #sRT_ConsecutiveCtrl.Q THEN
               "LBP_AlarmMsgs".UserA[03].A70UUxx[27] := TRUE;
           END_IF;
       END_IF;
   END_REGION
END_FUNCTION_BLOCK

FUNCTION_BLOCK "FB_LoaderShuttle1"   // FB204, SCL
{ S7_Optimized_Access := 'TRUE' }
// stored: AutoNumber false, MemoryReserve 100, SetENOAutomatically false
   VAR_INPUT
      iGripperReserved : Bool;
      iGripperReleased : Bool;
      iShuttleMoving : Bool;
      iShuttleInPos : Bool;
      iAxisV_Moving : Bool;
      iAxisV_InPos : Bool;
      iAxisW_Moving : Bool;
      iAxisW_InPos : Bool;
   END_VAR
   VAR_OUTPUT
      oExtGateOpenReq : Bool;
      oExtGateCloseReq : Bool;
      oIntGateOpenReq : Bool;
      oIntGateCloseReq : Bool;
      oLoadGripperCloseReq : Bool;
      oUnloadGripperOpenReq : Bool;
      oBlowingReq : Bool;
      oShuttleStartReq : Bool;
      oShuttlePosSetPoint : Real;
      oAxisVStartReq : Bool;
      oAxisVPosSetPoint : Real;
      oAxisWStartReq : Bool;
      oAxisWPosSetPoint : Real;
   END_VAR
   VAR
      sMain : "FB_Main";
      sShuttleInt { S7_SetPoint := 'True'} : "FB_ShuttleInt";
      sShuttleExt { S7_SetPoint := 'True'} : "FB_ShuttleExt";
      sControlIn { S7_SetPoint := 'True'} : "FB_PartControl";
      sControlOut { S7_SetPoint := 'True'} : "FB_PartControl";
      sBlowing { S7_SetPoint := 'True'} : "FB_Blowing";
      sIntLoadUnload { S7_SetPoint := 'True'} : "FB_IntLoadUnload";
      sExtLoadUnload { S7_SetPoint := 'True'} : "FB_ExtLoadUnload";
      sBwLoadUnload { S7_SetPoint := 'True'} : "FB_BwLoadUnload";
      sBwControlIn { S7_SetPoint := 'True'} : "FB_BwControl";
      sActPartControlIn { S7_SetPoint := 'True'} : "FB_ActControl";
      sActPartControlOut { S7_SetPoint := 'True'} : "FB_ActControl";
      sActBwControlIn { S7_SetPoint := 'True'} : "FB_ActControl";
      sIntLoadUnloadOP { S7_SetPoint := 'True'} : "FB_IntLoadUnloadOP";
      sBwConsecutiveCtrl { S7_SetPoint := 'True'} : "FB_Consecutive";
      sShuttlePosInt { S7_SetPoint := 'True'} : Bool;
      sShuttlePosSas : Bool;
      sShuttlePosExt : Bool;
      sGripper_OK : Bool;
      sExtLoaderInSafePos : Bool;
      sIntLoaderInSafePos : Bool;
      sBwLoaderInSafePos : Bool;
      sRT_PartControlInMissing : R_TRIG;
      sRT_PartControlInExtra : R_TRIG;
      sRT_PartControlOutMissing : R_TRIG;
      sRT_PartControlOutExtra : R_TRIG;
      sRT_BwControlInMissing : R_TRIG;
      sRT_BwControlInExtra : R_TRIG;
      sStepPauseSeq { S7_SetPoint := 'True'} : Bool;
   END_VAR
   VAR_TEMP
      tAxis_U_Position : Struct
         ExtLoadUnloadAuto : Bool;
         ExtLoadUnloadManu : Bool;
         PartControl : Bool;
         BwLoad : Bool;
         BwUnload : Bool;
         BwControl : Bool;
         IntLoadUnload : Bool;
         Blowing : Bool;
         IntLoadUnloadOP : Bool;
      END_STRUCT;
      tAxis_V_Position : Struct
         LoadUnload : Bool;
         Safe : Bool;
         Blowing : Bool;
      END_STRUCT;
      tAxis_W_Position : Struct
         LoadUnload : Bool;
         Safe : Bool;
         Approach : Bool;
         Blowing : Bool;
      END_STRUCT;
   END_VAR
BEGIN
   REGION Shuttle 1 position
       // Init Position
       #sShuttlePosInt := FALSE;
       #sShuttlePosSas := FALSE;
       #sShuttlePosExt := FALSE;

       // Check Shuttle (U1 Axis) position
       IF "DB_AxisPosition".sAxis05_U1."$AA_IM" < "DB_AxisPosMachinePLC".Axis_U1.IntGateExt THEN
           #sShuttlePosExt := TRUE;
       ELSIF "DB_AxisPosition".sAxis05_U1."$AA_IM" > "DB_AxisPosMachinePLC".Axis_U1.ExtGateInt THEN
           #sShuttlePosInt := TRUE;
       ELSE
           #sShuttlePosSas := TRUE;
       END_IF;
   END_REGION

   REGION Position Check
       REGION Axis U1
           // Position : External Load / Unload Auto
           "FC_PositionCheck"(iAxisCurrentPos := "DB_AxisPosition".sAxis05_U1."$AA_IM",
                              iAxisTargetPos := "DB_AxisPosMachinePLC".Axis_U1.ExtLoadUnloadAuto,
                              iTolMin := 0.001,
                              iTolMax := 0.001,
                              iInPos => #tAxis_U_Position.ExtLoadUnloadAuto);

           // Position : External Load / Unload Manu
           "FC_PositionCheck"(iAxisCurrentPos := "DB_AxisPosition".sAxis05_U1."$AA_IM",
                              iAxisTargetPos := "DB_AxisPosMachinePLC".Axis_U1.ExtLoadUnloadManu,
                              iTolMin := 0.001,
                              iTolMax := 0.001,
                              iInPos => #tAxis_U_Position.ExtLoadUnloadManu);

           // Position : Part Control
           "FC_PositionCheck"(iAxisCurrentPos := "DB_AxisPosition".sAxis05_U1."$AA_IM",
                              iAxisTargetPos := "DB_AxisPosMachinePLC".Axis_U1.PartControl,
                              iTolMin := 0.001,
                              iTolMax := 0.001,
                              iInPos => #tAxis_U_Position.PartControl);

           // Position : Backwall Load
           "FC_PositionCheck"(iAxisCurrentPos := "DB_AxisPosition".sAxis05_U1."$AA_IM",
                              iAxisTargetPos := "DB_AxisPosMachinePLC".Axis_U1.BwLoad,
                              iTolMin := 0.001,
                              iTolMax := 0.001,
                              iInPos => #tAxis_U_Position.BwLoad);

           // Position : Backwall Unload
           "FC_PositionCheck"(iAxisCurrentPos := "DB_AxisPosition".sAxis05_U1."$AA_IM",
                              iAxisTargetPos := "DB_AxisPosMachinePLC".Axis_U1.BwUnLoad,
                              iTolMin := 0.001,
                              iTolMax := 0.001,
                              iInPos => #tAxis_U_Position.BwUnload);

           // Position : Backwall Control
           "FC_PositionCheck"(iAxisCurrentPos := "DB_AxisPosition".sAxis05_U1."$AA_IM",
                              iAxisTargetPos := "DB_AxisPosMachinePLC".Axis_U1.BwControl,
                              iTolMin := 0.001,
                              iTolMax := 0.001,
                              iInPos => #tAxis_U_Position.BwControl);

           // Position : Internal Load / Unload
           "FC_PositionCheck"(iAxisCurrentPos := "DB_AxisPosition".sAxis05_U1."$AA_IM",
                              iAxisTargetPos := "DB_AxisPosMachinePLC".Axis_U1.IntLoadUnload,
                              iTolMin := 0.001,
                              iTolMax := 0.001,
                              iInPos => #tAxis_U_Position.IntLoadUnload);

           // Position : Internal Load / Unload OP
           "FC_PositionCheck"(iAxisCurrentPos := "DB_AxisPosition".sAxis05_U1."$AA_IM",
                              iAxisTargetPos := "DB_AxisPosMachinePLC".Axis_U1.IntLoadUnloadOP,
                              iTolMin := 0.001,
                              iTolMax := 0.001,
                              iInPos => #tAxis_U_Position.IntLoadUnloadOP);

           // Position : Blowing (Undrilled part)
           "FC_PositionCheck"(iAxisCurrentPos := "DB_AxisPosition".sAxis05_U1."$AA_IM",
                              iAxisTargetPos := "DB_AxisPosMachinePLC".Axis_U1.Blowing,
                              iTolMin := 0.001,
                              iTolMax := 0.001,
                              iInPos => #tAxis_U_Position.Blowing);
       END_REGION

       REGION Axis V
           // Position : Load / Unload Auto
           "FC_PositionCheck"(iAxisCurrentPos := "DB_AxisPosition".sAxis07_V."$AA_IM",
                              iAxisTargetPos := "DB_AxisPosMachinePLC".Axis_V.Shuttle_1.LoadUnload,
                              iTolMin := 0.001,
                              iTolMax := 0.001,
                              iInPos => #tAxis_V_Position.LoadUnload);

           // Position : Safe
           "FC_PositionCheck"(iAxisCurrentPos := "DB_AxisPosition".sAxis07_V."$AA_IM",
                              iAxisTargetPos := "DB_AxisPosMachinePLC".Axis_V.Safe,
                              iTolMin := 0.001,
                              iTolMax := 0.001,
                              iInPos => #tAxis_V_Position.Safe);

           // Position : Blowing
           "FC_PositionCheck"(iAxisCurrentPos := "DB_AxisPosition".sAxis07_V."$AA_IM",
                              iAxisTargetPos := "DB_AxisPosMachinePLC".Axis_V.Shuttle_1.Blowing,
                              iTolMin := 0.001,
                              iTolMax := 0.001,
                              iInPos => #tAxis_V_Position.Blowing);
       END_REGION

       REGION Axis W
           // Position : Load / Unload Auto
           "FC_PositionCheck"(iAxisCurrentPos := "DB_AxisPosition".sAxis08_W."$AA_IM",
                              iAxisTargetPos := "DB_AxisPosMachinePLC".Axis_W.Shuttle_1.LoadUnload,
                              iTolMin := 0.001,
                              iTolMax := 0.001,
                              iInPos => #tAxis_W_Position.LoadUnload);

           // Position : Safe
           "FC_PositionCheck"(iAxisCurrentPos := "DB_AxisPosition".sAxis08_W."$AA_IM",
                              iAxisTargetPos := "DB_AxisPosMachinePLC".Axis_W.Safe,
                              iTolMin := 0.001,
                              iTolMax := 0.001,
                              iInPos => #tAxis_W_Position.Safe);

           // Position : Approach (confondu avec load/unload)
           "FC_PositionCheck"(iAxisCurrentPos := "DB_AxisPosition".sAxis08_W."$AA_IM",
                              iAxisTargetPos := "DB_AxisPosMachinePLC".Axis_W.Shuttle_1.Approach,
                              iTolMin := 0.001,
                              iTolMax := 0.001,
                              iInPos => #tAxis_W_Position.Approach);

           // Position : Blowing
           "FC_PositionCheck"(iAxisCurrentPos := "DB_AxisPosition".sAxis08_W."$AA_IM",
                              iAxisTargetPos := "DB_AxisPosMachinePLC".Axis_W.Shuttle_1.Blowing,
                              iTolMin := 0.001,
                              iTolMax := 0.001,
                              iInPos => #tAxis_W_Position.Blowing);
       END_REGION
   END_REGION

   REGION Step Pause Sequence
       #sStepPauseSeq := "LBP_ModeGroup".E_JOG
       OR "DB_CycleStartStop".sResquestStopNextCycle
       OR "LBP_Chan1".E_M01;

       #sMain.iStepPause := #sStepPauseSeq;
       #sShuttleInt.iStepPause := #sStepPauseSeq;
       #sShuttleExt.iStepPause := #sStepPauseSeq;
       #sIntLoadUnload.iStepPause := #sStepPauseSeq;
       #sIntLoadUnloadOP.iStepPause := #sStepPauseSeq;
       #sControlIn.iStepPause := #sStepPauseSeq;
       #sControlOut.iStepPause := #sStepPauseSeq;
       #sBwLoadUnload.iStepPause := #sStepPauseSeq;
       #sBwControlIn.iStepPause := #sStepPauseSeq;
       #sBlowing.iStepPause := #sStepPauseSeq;
       #sActPartControlIn.iStepPause := FALSE;
       #sActPartControlOut.iStepPause := FALSE;
       #sActBwControlIn.iStepPause := FALSE;
   END_REGION

   REGION Main
       // Gripper prêt à Charger / Décharger une pièce
       #sGripper_OK :=
       (("DB_PartManagement".sPosition.sShuttle1.Undrilled.Presence.Part AND NOT "DB_PartManagement".sPosition.sGripper.Undrilled.Presence.Part AND "DB_GestionGripper".sUndrilledGripper.oStateOpen) OR NOT "DB_PartManagement".sPosition.sShuttle1.Undrilled.Presence.Part)
       AND (("DB_PartManagement".sPosition.sGripper.Drilled.Presence.Part AND NOT "DB_PartManagement".sPosition.sShuttle1.Drilled.Presence.Part) OR NOT "DB_PartManagement".sPosition.sGripper.Drilled.Presence.Part);

      // Loader INT in Safe Position
      #sIntLoaderInSafePos := "DB_AxisPosition".sAxis07_V."$AA_IM" >= "DB_AxisPosMachinePLC".Axis_V.Safe
      OR ("DB_AxisPosition".sAxis07_V."$AA_IM" < "DB_AxisPosMachinePLC".Axis_V.Safe AND "DB_AxisPosition".sAxis08_W."$AA_IM" >= "DB_AxisPosMachinePLC".Axis_W.Safe);

      // Loader EXT in Safe Position
      #sExtLoaderInSafePos := "DB_SonplasMain".sSonplasLoader.iOperateInOutCollision;

      // BW Loader in Safe Position
      #sBwLoaderInSafePos := "DB_BwLoaderExchange".Inputs.BwLoaderInSafePos;

      // Test Stop after Emptying with only one Shuttle
      IF ("DB_WorkingModes".sEmptying
          AND NOT "DB_LoaderShuttle2".sMain.iJobReq
          AND "DB_PartManagement".sPosition.sPartNumber.Total <= 1) THEN
          #sMain.iJobReq := FALSE;
      END_IF;
      // Test Stop after Emptying with two Shuttle
      IF ("DB_WorkingModes".sEmptying
          AND "DB_LoaderShuttle2".sMain.iJobReq
          AND #sMain.sCurrent_Step_NB =122
          AND "DB_PartManagement".sPosition.sPartNumber.Total <= 2) THEN
          #sMain.iJobReq := FALSE;
      END_IF;

      #sMain(iStartSeqCond := "DB_PowerOn".sMachineReadySoft AND NOT "MCP1_In".reset,
             iJobReq := #sMain.iJobReq,     
             iShuttleINT := #sShuttlePosInt,
             iShuttleSAS:= #sShuttlePosSas,
             iShuttleEXT := #sShuttlePosExt,
             iGripperReserved := #iGripperReserved,
             iGripperReleased := #iGripperReleased,
             iShuttleUndrilledPart:= "DB_PartManagement".sPosition.sShuttle1.Undrilled.Presence.Part,
             iShuttleDrilledPart:= "DB_PartManagement".sPosition.sShuttle1.Drilled.Presence.Part,
             iShuttleUndrilledBw:= "DB_PartManagement".sPosition.sShuttle1.Undrilled.Presence.BW,
             iShuttleDrilledBw:= "DB_PartManagement".sPosition.sShuttle1.Drilled.Presence.BW,
             iPartCtrlInOK:=#sControlIn.oPartControlOK,
             iPartCtrlInNOK:=#sControlIn.oPartControlNOK,
             iPartCtrlInContinuationStep:=#sActPartControlIn.oContinuationStep,
             iPartCtrlInRestartStep:=#sActPartControlIn.oRestartStep,
             iPartCtrlOutOK:=#sControlOut.oPartControlOK,
             iPartCtrlOutNOK:=#sControlOut.oPartControlNOK,
             iPartCtrlOutContinuationStep:=#sActPartControlOut.oContinuationStep,
             iPartCtrlOutRestartStep:=#sActPartControlOut.oRestartStep,
             iBwCtrlInOK:=#sBwControlIn.oBwControlOK,
             iBwCtrlInNOK:=#sBwControlIn.oBwControlNOK,
             iBwCtrlInContinuationStep:=#sActBwControlIn.oContinuationStep,
             iBwCtrlInRestartStep:=#sActBwControlIn.oRestartStep,
             iGripperOK:=#sGripper_OK,
             iNC_NoNeedAxis:= NOT "DB_CommPLC_ISO".sAxisManagedByNC,
             iExtLoaderInSafePos:=#sExtLoaderInSafePos,
             iIntLoaderInSafePos:=#sIntLoaderInSafePos,
             iBwLoaderInSafePos:=#sBwLoaderInSafePos,
             iOnePieceMode:="DB_WorkingModes".sOnePiece,
             iPLC_DateAndTime:= "DB_ReadDateAndTime".sDateAndTime,
             iStepPause:=#sMain.iStepPause,                                       
             oGripperAxisRequest => #sMain.oGripperAxisRequest,
             oGripperAxisRelease => #sMain.oGripperAxisRelease,
             oNoExtLoad=> #sMain.oNoExtLoad,
             oBwLoadReq=> #sMain.oBwLoadReq,
             oBwUnloadReq=> #sMain.oBwUnloadReq,
             ioShuttleIntSeq := #sShuttleInt.sInterface,
             ioShuttleExtSeq := #sShuttleExt.sInterface,
             ioControlInSeq := #sControlIn.sInterface,
             ioControlOutSeq := #sControlOut.sInterface,
             ioBlowingSeq:=#sBlowing.sInterface,
             ioIntLoadUnloadSeq := #sIntLoadUnload.sInterface,
             ioIntLoadUnloadOP_Seq:= #sIntLoadUnloadOP.sInterface,
             ioExtLoadUnloadSeq := #sExtLoadUnload.sInterface,
             ioBWLoadUnloadSeq := #sBwLoadUnload.sInterface,
             ioBWControlSeq := #sBwControlIn.sInterface,
             ioActPartControlInSeq:= #sActPartControlIn.sInterface,
             ioActPartControlOutSeq:= #sActPartControlOut.sInterface,
             ioActBwControlInSeq:= #sActBwControlIn.sInterface);
   END_REGION

   REGION Msg Sequence Fault
       // Msg 700014 Shuttle 1 Sequence Fault
       IF #sMain.sCurrent_Step_NB = 999 THEN
           "LBP_AlarmMsgs".UserA[00].A70UUxx[14] := TRUE;
       END_IF;
   END_REGION

   REGION Shuttle 1 INT
       // Position INT :
       //  IF Blowing : Pos. Blowing else Pos. Load/Unload
       IF "DB_LoaderOptions".Blowing.Disabled THEN
           #sShuttleInt.iShuttlePosIntSetPoint := "DB_AxisPosMachinePLC".Axis_U1.IntLoadUnload;
       ELSE
           #sShuttleInt.iShuttlePosIntSetPoint := "DB_AxisPosMachinePLC".Axis_U1.Blowing;
       END_IF;

       #sShuttleInt(iStartSeqCond := (#sMain.iStartSeqCond AND NOT #sShuttleInt.sInterface.Error AND NOT "DB_LoaderShuttle2".sShuttleInt.sInterface.SequenceRun AND #sShuttleInt.sInterface.StartRequest),
                    iJobReq := #sShuttleInt.sInterface.StartRequest,
                    iIntGateOpened := "DB_DigitalInputs".sInternalGateOpened.sSWStatus,
                    iIntGateClosed := "DB_DigitalInputs".sInternalGateLocked.sSWStatus,
                    iExtGateOpened := "DB_DigitalInputs".sExternalGateOpened.sSWStatus,
                    iExtGateClosed := "DB_DigitalInputs".sExternalGateLocked.sSWStatus,
                    iShuttlePosInt := #sShuttlePosInt,
                    iShuttlePosSas := #sShuttlePosSas,
                    iShuttlePosExt := #sShuttlePosExt,
                    iShuttlePosIntSetPoint := #sShuttleInt.iShuttlePosIntSetPoint,
                    iShuttlePosSasSetPoint := "DB_AxisPosMachinePLC".Axis_U1.Sas,
                    iShuttleMoving := #iShuttleMoving,
                    iShuttleInPos := #iShuttleInPos,
                    iIntLoaderInSafePos := #sIntLoaderInSafePos, 
                    iPLC_DateAndTime:= "DB_ReadDateAndTime".sDateAndTime,
                    iStepPause:=#sShuttleInt.iStepPause, 
                    oExtGateOpenReq => #sShuttleInt.oExtGateOpenReq,
                    oExtGateCloseReq => #sShuttleInt.oExtGateCloseReq,
                    oIntGateOpenReq => #sShuttleInt.oIntGateOpenReq,
                    oIntGateCloseReq => #sShuttleInt.oIntGateCloseReq,
                    oShuttleStartReq => #sShuttleInt.oShuttleStartReq,
                    oShuttlePosSetPoint => #sShuttleInt.oShuttlePosSetPoint);
   END_REGION

   REGION Shuttle 1 EXT
       #sShuttleExt(iStartSeqCond:= (#sIntLoaderInSafePos AND #sBwLoaderInSafePos AND #sMain.iStartSeqCond AND NOT #sShuttleExt.sInterface.Error AND NOT "DB_LoaderShuttle2".sShuttleExt.sInterface.SequenceRun AND #sShuttleExt.sInterface.StartRequest),
                    iJobReq:= #sShuttleExt.sInterface.StartRequest,
                    iIntGateOpened := "DB_DigitalInputs".sInternalGateOpened.sSWStatus,
                    iIntGateClosed := "DB_DigitalInputs".sInternalGateLocked.sSWStatus,
                    iExtGateOpened := "DB_DigitalInputs".sExternalGateOpened.sSWStatus,
                    iExtGateClosed := "DB_DigitalInputs".sExternalGateLocked.sSWStatus,
                    iShuttlePosInt:= #sShuttlePosInt,
                    iShuttlePosSas:= #sShuttlePosSas,
                    iShuttlePosExt:= #sShuttlePosExt,
                    iShuttlePosExtSetPoint:= "DB_AxisPosMachinePLC".Axis_U1.BwUnLoad,
                    iShuttlePosSasSetPoint:= "DB_AxisPosMachinePLC".Axis_U1.Sas,
                    iShuttleMoving := #iShuttleMoving,
                    iShuttleInPos := #iShuttleInPos,
                    iExtLoaderInSafePos:= #sExtLoaderInSafePos,
                    iPLC_DateAndTime:= "DB_ReadDateAndTime".sDateAndTime,
                    iStepPause:=#sShuttleExt.iStepPause,                 
                    oExtGateOpenReq => #sShuttleExt.oExtGateOpenReq,
                    oExtGateCloseReq => #sShuttleExt.oExtGateCloseReq,
                    oIntGateOpenReq => #sShuttleExt.oIntGateOpenReq,
                    oIntGateCloseReq => #sShuttleExt.oIntGateCloseReq,
                    oShuttleStartReq => #sShuttleExt.oShuttleStartReq,
                    oShuttlePosSetPoint => #sShuttleExt.oShuttlePosSetPoint);
   END_REGION

   REGION Ext_LoadUnload
       #sExtLoadUnload(iStartSeqCond := (#sExtLoaderInSafePos AND #sMain.iStartSeqCond AND NOT #sExtLoadUnload.sInterface.Error AND NOT "DB_LoaderShuttle2".sExtLoadUnload.sInterface.SequenceRun AND #sExtLoadUnload.sInterface.StartRequest AND #sShuttlePosExt),
                       iJobReq := #sExtLoadUnload.sInterface.StartRequest,
                       iShuttleExtLoadUnloadAutoPos := #tAxis_U_Position.ExtLoadUnloadAuto,
                       iShuttleExtLoadUnloadAutoPosSetPoint := "DB_AxisPosMachinePLC".Axis_U1.ExtLoadUnloadAuto,
                       iShuttleExtLoadUnloadManuPos := #tAxis_U_Position.ExtLoadUnloadManu,
                       iShuttleExtLoadUnloadManuPosSetPoint := "DB_AxisPosMachinePLC".Axis_U1.ExtLoadUnloadManu,
                       iShuttleMoving := #iShuttleMoving,
                       iShuttleInPos := #iShuttleInPos,
                       iCommunicationWithExtLoaderDone := "DB_SonplasMain".sSonplasLoader.iPartInShuttle1Finished,
                       iLoadUnloadMsgManuModeAck := #sExtLoadUnload.iLoadUnloadMsgManuModeAck OR "MCP1_In".plus OR "DI_SemiAutoValid", // WFA TBD
                       iAutoMode := "DB_WorkingModes".sAuto,
                       iSemiAutoMode := "DB_WorkingModes".sSemiAuto,
                       iFillingMode := "DB_WorkingModes".sFilling AND NOT #sMain.oNoExtLoad,
                       iEmptyingMode := "DB_WorkingModes".sEmptying OR #sMain.oNoExtLoad,
                       iPLC_DateAndTime:= "DB_ReadDateAndTime".sDateAndTime,
                       iStepPause:= #sExtLoadUnload.iStepPause,                 
                       oShuttleStartReq => #sExtLoadUnload.oShuttleStartReq,
                       oShuttlePosSetPoint => #sExtLoadUnload.oShuttlePosSetPoint,
                       oStartCommunicationWithExtLoader => "DB_SonplasMain".sSonplasLoader.oPartOutShuttle1InPos,
                       oSetLoadUnloadMsgManuMode => #sExtLoadUnload.oSetLoadUnloadMsgManuMode);    // WFA TBD

       // Message "Part loaded by operator"
       // IF #sExtLoadUnload.oSetLoadUnloadMsgManuMode THEN
       //     "LBP_AlarmMsgs".UserA[00].A70UUxx[55] := TRUE;
       // ELSIF
       //     #sExtLoadUnload.iLoadUnloadMsgManuModeAck OR "LBP_Chan1".A_Reset THEN
       //     "LBP_AlarmMsgs".UserA[00].A70UUxx[55] := FALSE;
       // END_IF;
       "LBP_AlarmMsgs".UserA[00].A70UUxx[55] := FALSE;
        #sExtLoadUnload.iLoadUnloadMsgManuModeAck := FALSE;
   END_REGION

   REGION Int_LoadUnload
       // Load Gripper Closed according to dry run working mode
        #sIntLoadUnload.iLoadGripperClosed := ("DB_GestionGripper".sUndrilledGripper.oStateCloseWithPart AND NOT "DB_WorkingModes".sDryRun)
        OR ("DB_GestionGripper".sUndrilledGripper.oStateClose AND "DB_WorkingModes".sDryRun);

       #sIntLoadUnload(iStartSeqCond := (#sIntLoaderInSafePos AND #sMain.iStartSeqCond AND NOT #sIntLoadUnload.sInterface.Error AND NOT "DB_LoaderShuttle2".sIntLoadUnload.sInterface.SequenceRun AND #sIntLoadUnload.sInterface.StartRequest AND #sShuttlePosInt),
                       iJobReq := #sIntLoadUnload.sInterface.StartRequest,
                       iShuttleIntLoadUnloadPos := #tAxis_U_Position.IntLoadUnload,
                       iShuttleIntLoadUnloadPosSetPoint := "DB_AxisPosMachinePLC".Axis_U1.IntLoadUnload,
                       iAxisV_LoadUnloadShuttlePos := #tAxis_V_Position.LoadUnload,
                       iAxisV_LoadUnloadShuttlePosSetPoint := "DB_AxisPosMachinePLC".Axis_V.Shuttle_1.LoadUnload,
                       iAxisV_SafePos := #tAxis_V_Position.Safe,
                       iAxisV_SafePosSetPoint := "DB_AxisPosMachinePLC".Axis_V.Safe,
                       iAxisW_SafePos := #tAxis_W_Position.Safe,
                       iAxisW_SafePosSetPoint := "DB_AxisPosMachinePLC".Axis_W.Safe,
                       iAxisW_ApproachLoadUnloadPos := #tAxis_W_Position.Approach,
                       iAxisW_ApproachLoadUnloadSetPoint := "DB_AxisPosMachinePLC".Axis_W.Shuttle_1.Approach,
                       iAxisW_LoadUnloadPos := #tAxis_W_Position.LoadUnload,
                       iAxisW_LoadUnloadPosSetPoint := "DB_AxisPosMachinePLC".Axis_W.Shuttle_1.LoadUnload,
                       iShuttleMoving := #iShuttleMoving,
                       iShuttleInPos := #iShuttleInPos,
                       iAxisV_Moving := #iAxisV_Moving,
                       iAxisV_InPos := #iAxisV_InPos,
                       iAxisW_Moving := #iAxisW_Moving,
                       iAxisW_InPos := #iAxisW_InPos,
                       iDrilledPartToUnload := "DB_PartManagement".sPosition.sGripper.Drilled.Presence.Part,
                       iUnDrilledPartToLoad := "DB_PartManagement".sPosition.sShuttle1.Undrilled.Presence.Part,
                       iLoadGripperClosed := #sIntLoadUnload.iLoadGripperClosed,
                       iUnloadGripperOpen := "DB_GestionGripper".sDrilledGripper.oStateOpen,
                       iPLC_DateAndTime := "DB_ReadDateAndTime".sDateAndTime,
                       iStepPause := #sIntLoadUnload.iStepPause,    
                       oShuttleStartReq => #sIntLoadUnload.oShuttleStartReq,
                       oShuttlePosSetPoint => #sIntLoadUnload.oShuttlePosSetPoint,
                       oAxisV_StartReq => #sIntLoadUnload.oAxisV_StartReq,
                       oAxisV_PosSetPoint => #sIntLoadUnload.oAxisV_PosSetPoint,
                       oAxisW_StartReq => #sIntLoadUnload.oAxisW_StartReq,
                       oAxisW_PosSetPoint => #sIntLoadUnload.oAxisW_PosSetPoint,
                       oLoadGripperCloseReq => #sIntLoadUnload.oLoadGripperCloseReq,
                       oUnloadGripperOpenReq => #sIntLoadUnload.oUnloadGripperOpenReq);
   END_REGION

   REGION Int_LoadUnloadOP
       // Load Gripper Closed according to dry run working mode
        #sIntLoadUnloadOP.iLoadGripperClosed := ("DB_GestionGripper".sUndrilledGripper.oStateCloseWithPart AND NOT "DB_WorkingModes".sDryRun)   // WFA A remettre
        OR ("DB_GestionGripper".sUndrilledGripper.oStateClose AND "DB_WorkingModes".sDryRun);

